// TIA Portal V17 program export: 1 tag tables, 17 data types, 25 data blocks, 3 code blocks (in call order from the OBs), 2 instance data blocks

VAR_GLOBAL   // PLC tag table "Default tag table"
   System_Byte AT %MB1000 : Byte;
   FirstScan AT %M1000.0 : Bool;
   DiagStatusUpdate AT %M1000.1 : Bool;
   AlwaysTRUE AT %M1000.2 : Bool;
   AlwaysFALSE AT %M1000.3 : Bool;
   Clock_Byte AT %MB1001 : Byte;
   Clock_10Hz AT %M1001.0 : Bool;
   Clock_5Hz AT %M1001.1 : Bool;
   "Clock_2.5Hz" AT %M1001.2 : Bool;
   Clock_2Hz AT %M1001.3 : Bool;
   "Clock_1.25Hz" AT %M1001.4 : Bool;
   Clock_1Hz AT %M1001.5 : Bool;
   "Clock_0.625Hz" AT %M1001.6 : Bool;
   "Clock_0.5Hz" AT %M1001.7 : Bool;
   TestReceive AT %M0.0 : Bool;
   ProductIn_Mem AT %M2.0 : LInt;
   GitTest AT %M0.1 : Bool;
END_VAR

TYPE "Speed_Change_Parameters"
// stored: IsFailsafeCompliant false
   STRUCT
      LabelSpeed : Int;   // Etikett hastighet
      IndexWheelVelocity : LReal;   // Indexhjul Hastighet
      IndexWheelAcceleration : LReal;   // Indexhjul Acceleration
      IndexWheelDeceleration : LReal;   // Indexhjul Decceration
      IndexWheelJerk : LReal;   // Indexhjul Jerk
   END_STRUCT;
END_TYPE

TYPE "UDT_Subsystem_Utility"
// stored: IsFailsafeCompliant false
   STRUCT
      Lifebit : Bool;   // Lifebit 1Hz, Check data exchange
      Fault : Bool;   // General Fault
      active : Bool;   // Machine is running or ready
      in_progress : Bool;   // Operation in is progress, motors are running
      EStop : Bool;   // Emergency stop active (1=good)
      General05 : Bool;   // General Signal, Operation mode 05
      General06 : Bool;   // General Signal, Operation mode 06
      General07 : Bool;   // General Signal, Operation mode 07
      General08 : Bool;   // General Signal, Operation mode 08
      General09 : Bool;   // General Signal, Operation mode 09
      General10 : Bool;   // General Signal, Operation mode 10
      General11 : Bool;   // General Signal, Operation mode 11
      General12 : Bool;   // General Signal, Operation mode 12
      General13 : Bool;   // General Signal, Operation mode 13
      General14 : Bool;   // General Signal, Operation mode 14
      General15 : Bool;   // General Signal, Operation mode 15
      Status00 : Bool;   // Motor running, status 00
      Status01 : Bool;   // Motor running, status 01
      Status02 : Bool;   // Motor running, status 02
      Status03 : Bool;   // Motor running, status 03
      Status04 : Bool;   // Motor running, status 04
      Status05 : Bool;   // Motor running, status 05
      Status06 : Bool;   // Motor running, status 06
      Status07 : Bool;   // Motor running, status 07
      Status08 : Bool;   // Motor running, status 08
      Status09 : Bool;   // Motor running, status 09
      Status10 : Bool;   // Motor running, status 10
      Status11 : Bool;   // Motor running, status 11
      Status12 : Bool;   // Motor running, status 12
      Status13 : Bool;   // Motor running, status 13
      Status14 : Bool;   // Motor running, status 14
      Status15 : Bool;   // Motor running, status 15
      Status16 : Bool;   // Motor running, status 16
      Status17 : Bool;   // Motor running, status 17
      Status18 : Bool;   // Motor running, status 18
      Status19 : Bool;   // Motor running, status 19
      Status20 : Bool;   // Motor running, status 20
      Status21 : Bool;   // Motor running, status 21
      Status22 : Bool;   // Motor running, status 22
      Status23 : Bool;   // Motor running, status 23
      Status24 : Bool;   // Motor running, status 24
      Status25 : Bool;   // Motor running, status 25
      Status26 : Bool;   // Motor running, status 26
      Status27 : Bool;   // Motor running, status 27
      Status28 : Bool;   // Motor running, status 28
      Status29 : Bool;   // Motor running, status 29
      Status30 : Bool;   // Motor running, status 30
      Status31 : Bool;   // Motor running, status 31
      Alarm000 : Bool;   // Alarm 0 active
      Alarm001 : Bool;   // Alarm 1 active
      Alarm002 : Bool;   // Alarm 2 active
      Alarm003 : Bool;   // Alarm 3 active
      Alarm004 : Bool;   // Alarm 4 active
      Alarm005 : Bool;   // Alarm 5 active
      Alarm006 : Bool;   // Alarm 6 active
      Alarm007 : Bool;   // Alarm 7 active
      Alarm008 : Bool;   // Alarm 8 active
      Alarm009 : Bool;   // Alarm 9 active
      Alarm010 : Bool;   // Alarm 10 active
      Alarm011 : Bool;   // Alarm 11 active
      Alarm012 : Bool;   // Alarm 12 active
      Alarm013 : Bool;   // Alarm 13 active
      Alarm014 : Bool;   // Alarm 14 active
      Alarm015 : Bool;   // Alarm 15 active
      Alarm016 : Bool;   // Alarm 16 active
      Alarm017 : Bool;   // Alarm 17 active
      Alarm018 : Bool;   // Alarm 18 active
      Alarm019 : Bool;   // Alarm 19 active
      Alarm020 : Bool;   // Alarm 20 active
      Alarm021 : Bool;   // Alarm 21 active
      Alarm022 : Bool;   // Alarm 22 active
      Alarm023 : Bool;   // Alarm 23 active
      Alarm024 : Bool;   // Alarm 24 active
      Alarm025 : Bool;   // Alarm 25 active
      Alarm026 : Bool;   // Alarm 26 active
      Alarm027 : Bool;   // Alarm 27 active
      Alarm028 : Bool;   // Alarm 28 active
      Alarm029 : Bool;   // Alarm 29 active
      Alarm030 : Bool;   // Alarm 30 active
      Alarm031 : Bool;   // Alarm 31 active
      Alarm032 : Bool;   // Alarm 32 active
      Alarm033 : Bool;   // Alarm 33 active
      Alarm034 : Bool;   // Alarm 34 active
      Alarm035 : Bool;   // Alarm 35 active
      Alarm036 : Bool;   // Alarm 36 active
      Alarm037 : Bool;   // Alarm 37 active
      Alarm038 : Bool;   // Alarm 38 active
      Alarm039 : Bool;   // Alarm 39 active
      Alarm040 : Bool;   // Alarm 40 active
      Alarm041 : Bool;   // Alarm 41 active
      Alarm042 : Bool;   // Alarm 42 active
      Alarm043 : Bool;   // Alarm 43 active
      Alarm044 : Bool;   // Alarm 44 active
      Alarm045 : Bool;   // Alarm 45 active
      Alarm046 : Bool;   // Alarm 46 active
      Alarm047 : Bool;   // Alarm 47 active
      Alarm048 : Bool;   // Alarm 48 active
      Alarm049 : Bool;   // Alarm 49 active
      Alarm050 : Bool;   // Alarm 50 active
      Alarm051 : Bool;   // Alarm 51 active
      Alarm052 : Bool;   // Alarm 52 active
      Alarm053 : Bool;   // Alarm 53 active
      Alarm054 : Bool;   // Alarm 54 active
      Alarm055 : Bool;   // Alarm 55 active
      Alarm056 : Bool;   // Alarm 56 active
      Alarm057 : Bool;   // Alarm 57 active
      Alarm058 : Bool;   // Alarm 58 active
      Alarm059 : Bool;   // Alarm 59 active
      Alarm060 : Bool;   // Alarm 60 active
      Alarm061 : Bool;   // Alarm 61 active
      Alarm062 : Bool;   // Alarm 62 active
      Alarm063 : Bool;   // Alarm 63 active
      Alarm064 : Bool;   // Alarm 64 active
      Alarm065 : Bool;   // Alarm 65 active
      Alarm066 : Bool;   // Alarm 66 active
      Alarm067 : Bool;   // Alarm 67 active
      Alarm068 : Bool;   // Alarm 68 active
      Alarm069 : Bool;   // Alarm 69 active
      Alarm070 : Bool;   // Alarm 70 active
      Alarm071 : Bool;   // Alarm 71 active
      Alarm072 : Bool;   // Alarm 72 active
      Alarm073 : Bool;   // Alarm 73 active
      Alarm074 : Bool;   // Alarm 74 active
      Alarm075 : Bool;   // Alarm 75 active
      Alarm076 : Bool;   // Alarm 76 active
      Alarm077 : Bool;   // Alarm 77 active
      Alarm078 : Bool;   // Alarm 78 active
      Alarm079 : Bool;   // Alarm 79 active
      Alarm080 : Bool;   // Alarm 80 active
      Alarm081 : Bool;   // Alarm 81 active
      Alarm082 : Bool;   // Alarm 82 active
      Alarm083 : Bool;   // Alarm 83 active
      Alarm084 : Bool;   // Alarm 84 active
      Alarm085 : Bool;   // Alarm 85 active
      Alarm086 : Bool;   // Alarm 86 active
      Alarm087 : Bool;   // Alarm 87 active
      Alarm088 : Bool;   // Alarm 88 active
      Alarm089 : Bool;   // Alarm 89 active
      Alarm090 : Bool;   // Alarm 90 active
      Alarm091 : Bool;   // Alarm 91 active
      Alarm092 : Bool;   // Alarm 92 active
      Alarm093 : Bool;   // Alarm 93 active
      Alarm094 : Bool;   // Alarm 94 active
      Alarm095 : Bool;   // Alarm 95 active
      Alarm096 : Bool;   // Alarm 96 active
      Alarm097 : Bool;   // Alarm 97 active
      Alarm098 : Bool;   // Alarm 98 active
      Alarm099 : Bool;   // Alarm 99 active
      Alarm100 : Bool;   // Alarm 100 active
      Alarm101 : Bool;   // Alarm 101 active
      Alarm102 : Bool;   // Alarm 102 active
      Alarm103 : Bool;   // Alarm 103 active
      Alarm104 : Bool;   // Alarm 104 active
      Alarm105 : Bool;   // Alarm 105 active
      Alarm106 : Bool;   // Alarm 106 active
      Alarm107 : Bool;   // Alarm 107 active
      Alarm108 : Bool;   // Alarm 108 active
      Alarm109 : Bool;   // Alarm 109 active
      Alarm110 : Bool;   // Alarm 110 active
      Alarm111 : Bool;   // Alarm 111 active
      Alarm112 : Bool;   // Alarm 112 active
      Alarm113 : Bool;   // Alarm 113 active
      Alarm114 : Bool;   // Alarm 114 active
      Alarm115 : Bool;   // Alarm 115 active
      Alarm116 : Bool;   // Alarm 116 active
      Alarm117 : Bool;   // Alarm 117 active
      Alarm118 : Bool;   // Alarm 118 active
      Alarm119 : Bool;   // Alarm 119 active
      Alarm120 : Bool;   // Alarm 120 active
      Alarm121 : Bool;   // Alarm 121 active
      Alarm122 : Bool;   // Alarm 122 active
      Alarm123 : Bool;   // Alarm 123 active
      Alarm124 : Bool;   // Alarm 124 active
      Alarm125 : Bool;   // Alarm 125 active
      Alarm126 : Bool;   // Alarm 126 active
      Alarm127 : Bool;   // Alarm 127 active
      OperatingHours : DWord;   // Operating hours of machine
      DownTimeHours : DWord;   // Downtime hours of machine
      Speed : Word;   // Production speed
      Container_total : DWord;   // Container counter of the actual batch.
      Container_good : DWord;   // Good container counter
      Container_reject : DWord;   // rejected container counter
      Counter_06 : DWord;   // Counter 06
      Counter_07 : DWord;   // Counter 07
      Counter_08 : DWord;   // Counter 08
      Counter_09 : DWord;   // Counter 09
      Counter_10 : DWord;   // Counter 10
      Counter_11 : DWord;   // Counter 11
      Total_Amount : Real;   // Total filling amount of the actual batch. [kg]
      Amount_01 : Real;   // Amount 01
      Amount_02 : Real;   // Amount 02
      Amount_03 : Real;   // Amount 03
      FormatName : String[20];
   END_STRUCT;
END_TYPE

TYPE "DataFromHSM"
// stored: IsFailsafeCompliant false
   STRUCT
      Sts : Struct
         xStop : Bool;   // Setzt den Spender in Stopp
         xRun : Bool;   // Setzt den Spender in Run
         xService : Bool;
         xTeach : Bool;
         xFeed : Bool;
         xConfigurationSave : Bool;
         xConfigurationLoad : Bool;
         xReceiveConfiguration : Bool;
         xCParameterSend : Bool;   // Schreibt alle über Kparam Maske ausgewählten Kparameter auf die ACP
         xCParameterReceive : Bool;   // Schreibt alle über Kparam Maske ausgewählten Kparameter in den DB
         xMparameterSend : Bool;   // Schreibt alle über Mparam Maske ausgewählten Mparameter auf die ACP
         xMparameterReceive : Bool;   // Schreibt alle über Mparam Maske ausgewählten parameter auf die DB
         xReserved : Bool;
         xGetTime : Bool;
         xGet_MAC_FW_version : Bool;
         xStatusContinuouslyTransmitted : Bool;   // 1: Aktiviert die kontinuierliche übertragung des Control Registers
         xCommunicationMonitoring : Bool;
         "x AcknowledgeFaultFromExternal" : Bool;
         xBlockProductSensor : Bool;   // 1: Produktsensor ist nicht aktiv, d.h. es wird kein Etikettierimpuls ausgelöst
         xSplice_Start : Bool;
         xReserved_25 : Bool;
         xReserved_24 : Bool;
         xReserved_23 : Bool;
         xReserved_22 : Bool;
         xReserved_21 : Bool;
         xReserved_20 : Bool;
         xReserved_19 : Bool;
         xReserved_18 : Bool;
         xReserved_17 : Bool;
         xReserved_16 : Bool;
         xReserved_15 : Bool;
         xReserved_14 : Bool;
         xDeviceStatusOK : Bool;
         xDeviceStatusWarning : Bool;
         xDeviceStatusAlarm : Bool;
         xPauseRun : Bool;
         xPauseStandby : Bool;
         xPauseService : Bool;
         xLampAlarm : Bool;
         xLampOK : Bool;
         xLampWarning : Bool;
         "xIO-Warning" : Bool;
         "xIO-Ready" : Bool;
         "xIO-Sync" : Bool;
         xSync2 : Bool;
         xSync3 : Bool;
         xLabelSensor : Bool;
         xProductSensorPolarity : Bool;
         xLowLabelSensor : Bool;
         xWebBreakSensor : Bool;
         xExternalStart : Bool;
         xSpliceActive : Bool;
         xReserved_12 : Bool;
         xReserved_11 : Bool;
         xReserved_10 : Bool;
         xReserved_09 : Bool;
         xReserved_08 : Bool;
         xReserved_07 : Bool;
         xReserved_06 : Bool;
         xReserved_05 : Bool;
         xReserved_04 : Bool;
         xReserved_03 : Bool;
         xReserved_02 : Bool;
         xReserved_01 : Bool;
         iLabelCounter : Int;
         iCounterRemaining : Int;
         iMcurr : Int;   // Status- Mittlerer Motorstrom in %
         wExtEncoder : Word;   // Status- Zählerwert des Ext. Encoders
         wErrorCode : Word;   // Fehlerwert
         wWarnNr : Word;   // Warnungscodes
         iReserved_W1 : Int;
         iReserved_W2 : Int;
         iReserved_W3 : Int;
         iReserved_W4 : Int;
         iReserved_W5 : Int;
         iReserved_W6 : Int;
      END_STRUCT;
      Cfg : Struct
         iLabellingSpeed : Int;   // in 1/10 m/min
         iTriggerDelay : Int;   // in 1/10 mm
         iLabelPosition : Int;   // in 1/10 mm
         iLabelLenght : Int;   // in mm
         iLabelGap : Int;   // in 1/10 mm
         iLabelsBurst : Int;   // 1=Aus, 2=zweimal … (mehrere Etiketten mit einem Triggerimpuls)
         iDistanceBetweenLabels : Int;   // in 1/10 mm (Abstand zwischen den Etiketten wenn mehrere pro Trigger)
         iMaxNumberOfLabelsToSkip : Int;   // 0 - n
         iTriggerBlank : Int;   // in mm
         iAccelerationRamp : Int;   // in 1/10 mm
         iSpeedInternalEncoder : Int;   // 0 = Intern, 1 = Drehgeber
         iStopRamp : Int;   // in % (Verhältnis zur Startrampe)
         iSyncOutputDelay : Int;   // in 1/10 mm
         iSyncOutputLength : Int;   // in 1/10 mm
         iSyncOutputDelay2 : Int;   // in 1/10 mm
         iSyncOutputLenght_2 : Int;   // in 1/10 mm
         iSyncOutputDelay_3 : Int;   // in 1/10 mm
         iSyncOutputLenght_3 : Int;   // in 1/10 mm
         iPreFeed : Int;   // in 1/10 mm
         iConveyorSpeed_1 : Int;
         iConveyorSpeed_2 : Int;
         iReserved_11 : Int;
         iReserved_10 : Int;
         iReserved_09 : Int;
         iReserved_08 : Int;
         iReserved_07 : Int;
         iReserved_06 : Int;
         iReserved_05 : Int;
         iReserved_04 : Int;
         iReserved_03 : Int;
         iReserved_02 : Int;
         iReserved_01 : Int;
      END_STRUCT;
      M_Par : Struct
         iSpeedInternalEncoder : Int;   // 0 = Fixed internally, 1 = Encoder fixed, 2 = Value from configuration
         iEncoderMMPerRevolution : Int;   // in 1/10 mm
         iEncoderPulsesPerRevolution : Int;   // in Pulse
         iMaximumSpeed : Int;   // in 1/10 m/min
         iInstallationMode : Int;   // 0 = normal, 1 = feed also via start button, 2 = feed with fixed length via start button, 3 = feed always with fixed length
         iLabelLengthInMMPerMotorRevolution : Int;   // in 1/100 mm
         iDistanceGapSensorToDispensingEdge : Int;   // in 1/10 mm
         iProductSensorPolarity : Int;   // 0 = NPN, 1 = NPN inverted, 2 = PNP inverted, 3 = PNP
         iSkipMode_1 : Int;   // 0 = value from configuration, 1 = value from machine parameters, 2 = end detect
         iMaxLabelSkip : Int;   // 0 - n
         iAccelerationMode : Int;   // 0 = value from configuration, 1 = value from machine parameters
         iAcceleration : Int;   // in 1/10 mm
         iGapSensor : Int;   // 0 = leading edge, 1 = trailing edge label
         iMaxCalibrationLength : Int;   // in 1/10mm
         iDecelarationMode : Int;   // 0 = value from configuration, 1 = value from machine parameters
         iDecelaration : Int;   // in % (of acceleration distance)
         iExernalStart : Int;   // 0 = off 1 = edge controlled 2 = pulse controlled
         iLowLabelInput : Int;   // 0= Off 1=On
         iBeltInput_1 : Int;   // 0= Off 1=On
         iSyncParameter_1 : Int;   // 0 = value from configuration, 1 = value from machine parameters
         iSyncOutputDelay : Int;   // in 1/10mm
         iSyncOutputLength : Int;   // in 1/10mm
         iZeroDownTimeMode_1 : Int;   // 0 = off 1 = master 2 = slave
         iZeroDownTimeSensorDistance : Int;   // in mm
         iLabelLengthInCaseOfErrorOnLowLabelSensor : Int;   // in m
         iLowLabelSensorPolarity : Int;   // 2 = PNP inverted 3 = PNP
         iWebBreakSensorPolarity : Int;   // 2 = PNP inverted 3 = PNP
         iWarningOutputPolarity_1 : Int;   // 2 = PNP inverted 3 = PNP
         iSync2Parameter_1 : Int;   // 0 = value from configuration, 1 = value from machine parameters
         iSync2OutputDelay_1 : Int;   // in 1/10mm
         iSync2OutputPulseLength_1 : Int;   // in 1/10mm
         iSync3Parameter_1 : Int;   // 0 = value from configuration, 1 = value from machine parameters
         iSync3OutputDelay_1 : Int;   // in 1/10mm
         iSync3OutputPulseLength_1 : Int;   // in 1/10mm
         iTeachTolerance : Int;   // in 1/100mm
         iSynch1Mode_1 : Int;   // 0 = production sensor 1 = trigger sensor 2 = reserve 3 = end of dispensing
         iSynch2Mode_1 : Int;   // 0 = production sensor 1 = trigger sensor 2 = reserve 3 = end of dispensing
         iSynch3Mode_1 : Int;   // 0 = production sensor 1 = trigger sensor 2 = reserve 3 = end of dispensing
         iOvercurrentCorrection : Int;   // in %
         iServiceFeedSpeed : Int;   // in 1/10 m/min
         iPreDispensingMode : Int;   // 0 = value from configuration, 1 = value from machine parameters
         iPreDispensingLength : Int;   // in 1/10 mm
         iLabelSensorWindowPreDispensingPath : Int;   // in 1/10 mm
         iLabelSensorCount : Int;
         "iSPS-Mode_1" : Int;   // 0 = Off 1 = S7 communication / 0= Off 1= S7-communication, 2 = S7-communication double size
         iZdtWin_1 : Int;   // Zero down time window mm / Zero Down Time Window mm
         iDistRes_1 : Int;   // Resolution label spacing
         "iSPS-DB-NoCtrl_1" : Int;   // SPS-DB-Nr Control (SPS->ACP) / Data block for PLC communication
         "iSPS-DB-NoStat_1" : Int;   // SPS-DB-Nr Status (ACP->SPS) / Data block for PLC communication
         iSignalFormat_1 : Int;   // Status-Server: Signalform / Is relevant for the WEBER-TOOL
         iLowLabDiam_1 : Int;   // Roll diameter for LowLabel in 1/10 mm / Roll diameter for LowLab in 1/10 mm
         iCoreDiameter_1 : Int;   // Core diameter in 1/10 mm
         iWebBreakRest_1 : Int;   // Rest after WebBreak in mm
         iLeverSetup_1 : Int;   // Do not use here / To the TEACH of the dancer position
         iLeverMinPos_1 : Int;   // Analog value angle sensor unwinder dancer Min.Pos.
         iLeverMaxPos_1 : Int;   // Analog value angle sensor unwinder dancer Max.Pos.
         "iUW-BufLength_1" : Int;   // Label path in mm between dancers min / max
         iTwinLabelMd_1 : Int;   // Double Label Mode / Double Label mode
         iLabelQueTolerans : Int;   // Setting the tolerance "Number of labels between peel bar and label sensor".
         iResetEvents : Int;   // Reset the operating data EV#007 „Number of all spent labels“ or EV#008 „Display of label roll dispensed“. 0 = off, 1 = reset EV#007 Label feeds, 2 = reset EV#008 Label meters.
         iMaintenanceDistanceKm : Int;   // Setting the maintenance interval depending on the the label roll length. [km]
         iMaintenanceDays : Int;   // Setting the maintenance interval depending on the operation time. [days]
         iProductSensorMode : Int;   // Defines the linkage of the product sensors 1 and 2 with respect to the trigger signal. 0 = Off, 1 = AND Operation (both sensors must recieve a signal), 2 = OR operation (only one sensor have to recieve a signal)
         iRewinderDiameterWarning : Int;   // Defines the diameter of the carrier web, after which a pre-warning for the rewinder is avti-vated. The following message appears "Rewinder almost full".
         arrayFirmwareVersion_1 : Array[0..19] of Char;   // Defines the diameter of the carrier web, after which the labeler stops. The following mes-sage appears "Rewinder full".
         "arrayCfg_MAC-Adress_1" : Array[0..19] of Char;   // Defines the value for the motor current, after which the following message appears "Load approaching the upper limit".
         iRewinderDiameterFull : Int;   // Parameter for activating contour mode. When the parameter is activated, the two parameters "Start contour" and "Stop contour" are displayed in the configuration menu. At the same time, the "Ramp" parameter is ignored.
         iMotorLoadLimit : Int;   // Determines the number of encoder pulses per millimeter of label path and synchronizes an optional printer at the AUX socket.
         iCountorRamp : Int;   // This Parameter is used to set the communication with different PLC versions.
         iEncoderOutPulsMM : Int;   // This parameter is used to set the distance (duration) in splice mode. The label web is ad-vanced with the reduced speed specified in parameter 071. 0 - 9999. Adjusting the value in [mm]
         iSPS_RackAndSlot : Int;   // This parameter is only used if parameter 070 is active. It is used to reduce reduce the speed in the slice mode and is calculated on the basis of the current speed. 10 - 100. Adjusting the value in [%]
         iSpliceDistance : Int;   // This parameter is only used for alternating operation and defines the transfer reserve that is still to be dispensed in alternating operation. Must be less than or equal to Par.25 RestLowLabel. 0.0 – 90.0. Adjusting the value in [m]
         iSpliceSpeedReduction : Int;   // Offset setting for operation with rotary encoder. The feed rate of the dispenser is factor Par.73 x encoder speed. 20.0 - 500.0. Adjusting the value in [%].
         iDownstream : Int := 20;   // Setting of the start ramp setting in m/s2. If the value is 0, the ramp length is used to calcu-late the acceleration. The stop ramp is set exactly as before via the ratio to the start ramp. 0.0 - 90.0. In [m/s2]
         iSpeedFactor : Int := 1000;   // Setting of a speed offset in 1/10 m/min. Only applies to the internal speed. Parameter 073 can be used in encoder mode. -20.0 - 20.0. in [%]
         iAcceleration_1 : Int := 0;   // Determines whether the material transport error "Materialtransportoffen" is to be output. The signal for the error must be applied to X22.4. 0 = Off. 1 = Error at 24V. 2 = Error at 0V.
         iSpeedOffset : Int := 0;   // Offset setting of the encoder speed for the internal calculation of Alpha HSM, e.g. for win-ding tape operation and ZDT application. Alpha HSM must calculate with baseband speed for the function of the ZDT, but dispenses with encoder speed from the winding belt. 20.0 - 500.0. In [%]
         iMaterialTransportErrorMode : Int := 0;   // Determines whether the material transport error "Materialtransportoffen" is to be output. The signal for the error must be applied to X22.4. 0 = Off. 1 = Error at 24V. 2 = Error at 0V.
         iEncoderFactor : Int := 1000;   // Offset setting of the encoder speed for the internal calculation of Alpha HSM, e.g. for win-ding tape operation and ZDT application. Alpha HSM must calculate with baseband speed for the function of the ZDT, but dispenses with encoder speed from the winding belt. 20.0 - 500.0. In [%]
         iReserve_1 : Int;
         iReserve_2 : Int;
         iReserve_3 : Int;
         iReserve_4 : Int;
         iReserve_5 : Int;
         iReserve_6 : Int;
         iReserve_7 : Int;
         iReserve_8 : Int;
         iReserve_9 : Int;
         iReserve_10 : Int;
         iReserve_11 : Int;
         iReserve_12 : Int;
         iReserve_13 : Int;
         iReserve_14 : Int;
         iReserve_15 : Int;
         iReserve_16 : Int;
         iReserve_17 : Int;
         iReserve_18 : Int;
         iReserve_19 : Int;
         iReserve_20 : Int;
         iReserve_21 : Int;
         iReserve_22 : Int;
         iReserve_23 : Int;
         iReserve_24 : Int;
         iReserve_25 : Int;
         iReserve_26 : Int;
         iReserve_27 : Int;
         iReserve_28 : Int;
         iReserve_29 : Int;
         iReserve_30 : Int;
         iReserve_31 : Int;
         iReserve_32 : Int;
         iReserve_33 : Int;
         iReserve_34 : Int;
         iReserve_35 : Int;
         iReserve_36 : Int;
         iReserve_37 : Int;
         iReserve_38 : Int;
         iReserve_39 : Int;
         iReserve_40 : Int;
         iReserve_41 : Int;
         iReserve_42 : Int;
         iReserve_43 : Int;
         iReserve_44 : Int;
         iReserve_45 : Int;
         iReserve_46 : Int;
         iReserve_47 : Int;
         iReserve_48 : Int;
         iReserve_49 : Int;
         iReserve_50 : Int;
         iReserve_51 : Int;
      END_STRUCT;
   END_STRUCT;
END_TYPE

TYPE "DataToHSM"
// stored: IsFailsafeCompliant false
   STRUCT
      Cmd : Struct   // Command Send
         xStop : Bool;   // Offline
         xRun : Bool;   // Online
         xService : Bool;
         xTeach : Bool;
         xFeed : Bool;
         xSaveConfiguration : Bool;   // Reserved but not used for the time being
         xLoadConfiguration : Bool;   // Reserved but not used for the time being
         xRecieveContent : Bool;   // Reserved but not used for the time being
         xCparameterSend : Bool;   // Starts sending all K parameters selected via Kparameter mask to the labeling system / Starts sending all C parameters selected via C parameter mask to the labeling system
         xCparameterReceive : Bool;   // Requests the labeling system to send all parameters
         xMparameterSend : Bool;   // Starts sending all the M parameters selected via the Mparameter mask to the labeling system
         xMparameterReceive : Bool;   // Requests all labeling parameters to be sent from the labeling system
         xReserve : Bool;
         xReceiveTime : Bool;
         xGetMACandFWversion : Bool;
         xActivateContinuousStatus : Bool;   // 1: Activates the continuous transfer of the control register (initially not used)
         xWatchDog : Bool;   // Sign of Life Bit
         xAcknowledgeFaultFromExternal : Bool;   // PLC can directly acknowledge a malfunction of the labeling system
         xBlockProductPhotocell : Bool;   // 1: Product sensor is not active, i.e. no labeling pulse is triggered
         "xSplice-Start" : Bool;
         xReserved_19 : Bool;
         xReserved_18 : Bool;
         xReserved_17 : Bool;
         xReserved_16 : Bool;
         xReserved_15 : Bool;
         xReserved_14 : Bool;
         xReserved_13 : Bool;
         xReserved_12 : Bool;
         xReserved_11 : Bool;
         xReserved_10 : Bool;
         xReserved_09 : Bool;
         xReserved_08 : Bool;
         ParaMask : "HSMConfigAndMachineParameterMask";
         iUpdateRate : Int;   // Rate in ms at which the control register is updated
         iReserved_03 : Int;
         iReserved_02 : Int;
         iReserved_01 : Int;
      END_STRUCT;
      Cfg : Struct   // Configuration Parameters Send
         iDesiredInternalSpeed : Int;   // in 1/10 m / min (desired speed value)
         iDispenseDelay : Int;   // in 1/10 mm
         iLabelPosition : Int;   // in 1/10 mm
         iLabelLength : Int;   // in mm
         iLabelGap : Int;   // in 1/10 mm
         iLabelBurst : Int;   // 1 = off, 2 = twice ... (several labels with one trigger pulse)
         iLabelDistance : Int;   // in 1/10 mm (distance between the labels if several per trigger)
         iMaxNumberOfLabelSkips : Int;   // 0 - n
         iTriggerBlanking : Int;   // in mm
         iAccelerationRamp : Int;   // in 1/10 mm
         iSpeedInternalOrEncoder : Int;   // 0 = internal, 1 = encoder
         iStopRamp : Int;   // in% (ratio to acceleration ramp)
         iSyncOutputDelay : Int;   // in 1/10 mm
         iSyncOutputLenght : Int;   // in 1/10 mm
         iSyncOutput2Delay : Int;   // in 1/10 mm
         iSyncOutput2Lenght : Int;   // in 1/10 mm
         iSyncOutput3Delay : Int;   // in 1/10 mm
         iSyncOutput3Lenght : Int;   // in 1/10 mm
         iPreFeedLenght : Int;   // in 1/10 mm
         iConveyorSpeed_1 : Int;
         iConveyorSpeed_2 : Int;
         iReserved_11 : Int;
         iReserved_10 : Int;
         iReserved_09 : Int;
         iReserved_08 : Int;
         iReserved_07 : Int;
         iReserved_06 : Int;
         iReserved_05 : Int;
         iReserved_04 : Int;
         iReserved_03 : Int;
         iReserved_02 : Int;
         iReserved_01 : Int;
      END_STRUCT;
      MPar : Struct   // Machine Parameters Send
         iSpeedInternalOrEncoder : Int;   // 0 = Fixed internally, 1 = Encoder fixed, 2 = Value from configuration
         iDistancePerEncoderRevolution : Int;   // in 1/10 mm
         iPulsesPerEncoderRevolution : Int;   // in Pulse
         iMaxSpeed : Int;   // in 1/10 m/min
         iInstallationsMode : Int;   // 0 = normal, 1 = feed also via start button, 2 = feed with fixed length via start button, 3 = feed always with fixed length
         iBackingPaperLengthPerMotorRevolution : Int;   // in 1/100 mm
         iDistanceToDispensingEdgeToGapSensor : Int;   // in 1/10 mm (required for changeable dispense tongues and changed depending on the product)
         iProductsensorPolarity : Int;   // 0 = NPN, 1 = NPN inverted, 2 = PNP inverted, 3 = PNP
         iSkipMode : Int;   // 0 = value from configuration, 1 = value from machine parameters, 2 = end detect
         iMaxNumberOfLabelSkips : Int;   // 0 - n
         iAccelerationRampMode : Int;   // 0 = value from configuration, 1 = value from machine parameters
         iAccelerationRamp : Int;   // in 1/10 mm
         iGapSensor : Int;   // 0 = leading edge, 1 = trailing edge label
         iMaxCalibrationDistance : Int;   // in 1/10mm
         iDecelerationRampMode : Int;   // 0 = value from configuration, 1 = value from machine parameters
         iDecelerationRamp : Int;   // in% (ratio to acceleration ramp)
         iExternalStart : Int;   // 0 = off 1 = edge controlled 2 = pulse controlled
         iLowLabelInput : Int;   // 0 = off 1 = on
         iRibbonInput : Int;   // 0 = off 1 = on
         iSyncParameter : Int;   // 0 = value from configuration, 1 = value from machine parameters
         iSyncOutputDelay : Int;   // in 1/10mm
         iSyncOutputLenght : Int;   // in 1/10mm
         iZeroDownTimeMode : Int;   // 0 = Off 1 = Master 2 = Slave
         iZeroDownTimeSensorDistance : Int;   // in mm
         iRestLenghtOnLowLabel : Int;   // in m
         iLowLabelSensorPolarity : Int;   // 2 = PNP inverted 3 = PNP
         iWebBreakSensorPolarity : Int;   // 2 = PNP inverted 3 = PNP
         iWarningOutputPolarity : Int;   // 2 = PNP inverted 3 = PNP
         iSync2Parameter : Int;   // 0 = value from configuration, 1 = value from machine parameters
         iSync2OutputDelay : Int;   // in 1/10mm
         iSync2OutputLenght : Int;   // in 1/10mm
         iSync3Parameter : Int;   // 0 = value from configuration, 1 = value from machine parameters
         iSync3OutputDelay : Int;   // in 1/10mm
         iSync3OutputLenght : Int;   // in 1/10mm
         iTeachTolerance : Int;   // in 1/100mm
         iSynch1Mode : Int;   // 0 = production sensor 1 = trigger sensor 2 = reserve 3 = end of dispense
         iSynch2Mode : Int;   // 0 = production sensor 1 = trigger sensor 2 = reserve 3 = end of dispense
         iSynch3Mode : Int;   // 0 = production sensor 1 = trigger sensor 2 = reserve 3 = end of dispense
         iOverCurrentCorrection : Int;   // in %
         iServiceFeedRate : Int := 10;   // in 1/10 m/min
         iPreFeedMode : Int;   // 0 = value from configuration, 1 = value from machine parameters
         iPreFeed : Int;   // in 1/10 mm
         iLabelSensorWindowPreFeedLenght : Int;   // in 1/10 mm
         iLabelSensorCount : Int;
         "iSPS-Mode" : Int;   // 0= Off 1= S7-Kommunikation / 0= Off 1= S7-communication, 2 = S7-communication double size
         iZdtWin : Int;   // Zero Down Time Window mm
         iDistRes : Int;   // Resolution label spacing
         "iSPS-DB-No-Ctrl" : Int;   // Data block for PLC communication
         "iSPS-DB-No-Stat" : Int;   // Data block for PLC communication
         iSignalFormat : Int;   // Is relevant for the WEBER-TOOL
         iLowLabDiam : Int;   // Roll diameter for LowLab in 1/10 mm
         iCoreDiameter : Int;   // Core diameter in 1/10 mm
         iWebBreakRest : Int;   // Rest after WebBreak in mm
         iLeverSetup : Int;   // To the TEACH of the dancer position
         iLeverMinPos : Int;   // Analog value angle sensor unwinder dancer Min.Pos.
         iLeverMaxPos : Int;   // Analog value angle sensor unwinder dancer Max.Pos.
         "iUW-BufLength" : Int;   // Label path in mm between dancers min / max
         iTwinLabelMd : Int;   // Double Label mode
         iLabQueuwTolerance : Int := 10;   // Setting the tolerance "Number of labels between peel bar and label sensor".
         iResetEvents : Int;   // Reset the operating data EV#007 „Number of all spent labels“ or EV#008 „Display of label roll dispensed“. 0 = off, 1 = reset EV#007 Label feeds, 2 = reset EV#008 Label meters.
         iMaintananceDistancekm : Int;   // Setting the maintenance interval depending on the the label roll length. [km]
         iMaintananceDays : Int;   // Setting the maintenance interval depending on the operation time. [days]
         iProductSensorMode : Int;   // Defines the linkage of the product sensors 1 and 2 with respect to the trigger signal. 0 = Off, 1 = AND Operation (both sensors must recieve a signal), 2 = OR operation (only one sensor have to recieve a signal)
         iRewinderDiameterWarning : Int := 2600;   // Defines the diameter of the carrier web, after which a pre-warning for the rewinder is avti-vated. The following message appears "Rewinder almost full".
         iRewinderDiameterFull : Int := 2650;   // Defines the diameter of the carrier web, after which the labeler stops. The following mes-sage appears "Rewinder full".
         iMotorLoadLimit : Int := 90;   // Defines the value for the motor current, after which the following message appears "Load approaching the upper limit".
         iContourRamp : Int;   // Parameter for activating contour mode. When the parameter is activated, the two parameters "Start contour" and "Stop contour" are displayed in the configuration menu. At the same time, the "Ramp" parameter is ignored.
         iEncoderOutPulsPermm : Int;   // Determines the number of encoder pulses per millimeter of label path and synchronizes an optional printer at the AUX socket.
         iPLCRackAndSlot : Int := 10;   // This Parameter is used to set the communication with different PLC versions.
         iSliceDistance : Int := 2000;   // This parameter is used to set the distance (duration) in splice mode. The label web is ad-vanced with the reduced speed specified in parameter 071. 0 - 9999. Adjusting the value in [mm]
         iSpliceSpeedReduction : Int := 33;   // This parameter is only used if parameter 070 is active. It is used to reduce reduce the speed in the slice mode and is calculated on the basis of the current speed. 10 - 100. Adjusting the value in [%]
         iDownstream : Int := 20;   // This parameter is only used for alternating operation and defines the transfer reserve that is still to be dispensed in alternating operation. Must be less than or equal to Par.25 RestLowLabel. 0.0 – 90.0. Adjusting the value in [m]
         iSpeedFactor : Int := 1000;   // Offset setting for operation with rotary encoder. The feed rate of the dispenser is factor Par.73 x encoder speed. 20.0 - 500.0. Adjusting the value in [%].
         iAcceleration : Int;   // Setting of the start ramp setting in m/s2. If the value is 0, the ramp length is used to calcu-late the acceleration. The stop ramp is set exactly as before via the ratio to the start ramp. 0.0 - 90.0. In [m/s2]
         iSpeedOffset : Int;   // Setting of a speed offset in 1/10 m/min. Only applies to the internal speed. Parameter 073 can be used in encoder mode. -20.0 - 20.0. in [%]
         iMaterialTransportErrorMode : Int;   // Determines whether the material transport error "Materialtransportoffen" is to be output. The signal for the error must be applied to X22.4. 0 = Off. 1 = Error at 24V. 2 = Error at 0V.
         iEncoderFactor : Int := 1000;   // Offset setting of the encoder speed for the internal calculation of Alpha HSM, e.g. for win-ding tape operation and ZDT application. Alpha HSM must calculate with baseband speed for the function of the ZDT, but dispenses with encoder speed from the winding belt. 20.0 - 500.0. In [%]
         Reserve_1 : Int;
         Reserve_2 : Int;
         Reserve_3 : Int;
         Reserve_4 : Int;
         Reserve_5 : Int;
         Reserve_6 : Int;
         Reserve_7 : Int;
         Reserve_8 : Int;
         Reserve_9 : Int;
         Reserve_10 : Int;
         Reserve_11 : Int;
         Reserve_12 : Int;
         Reserve_13 : Int;
         Reserve_14 : Int;
         Reserve_15 : Int;
         Reserve_16 : Int;
         Reserve_17 : Int;
         Reserve_18 : Int;
         Reserve_19 : Int;
         Reserve_20 : Int;
         Reserve_21 : Int;
         Reserve_22 : Int;
         Reserve_23 : Int;
         Reserve_24 : Int;
         Reserve_25 : Int;
         Reserve_26 : Int;
         Reserve_27 : Int;
         Reserve_28 : Int;
         Reserve_29 : Int;
         Reserve_30 : Int;
         Reserve_31 : Int;
         Reserve_32 : Int;
         Reserve_33 : Int;
         Reserve_34 : Int;
         Reserve_35 : Int;
         Reserve_36 : Int;
         Reserve_37 : Int;
         Reserve_38 : Int;
         Reserve_39 : Int;
         Reserve_40 : Int;
         Reserve_41 : Int;
         Reserve_42 : Int;
         Reserve_43 : Int;
         Reserve_44 : Int;
         Reserve_45 : Int;
         Reserve_46 : Int;
         Reserve_47 : Int;
         Reserve_48 : Int;
         Reserve_49 : Int;
         Reserve_50 : Int;
         Reserve_51 : Int;
      END_STRUCT;
   END_STRUCT;
END_TYPE

TYPE "HSMConfigAndMachineParameterMask"
// stored: IsFailsafeCompliant false
   STRUCT
      HSMConfig_1 : "HSMConfigParaMask1";
      HSMConfig_2 : "HSMConfigParaMask2";
      HSMMachine_1 { S7_SetPoint := 'True'} : "HSMMachineParaMask1";
      HSMMachine_2 { S7_SetPoint := 'True'} : "HSMMachineParaMask2";
      HSMMachine_3 { S7_SetPoint := 'True'} : "HSMMachineParaMask3";
      HSMMachine_4 { S7_SetPoint := 'True'} : "HSMMachineParaMask4";
      HSMMachine_5 { S7_SetPoint := 'True'} : "HSMMachineParaMask5";
      HSMMachine_6 { S7_SetPoint := 'True'} : "HSMMachineParaMask6";
      HSMMachine_7 { S7_SetPoint := 'True'} : "HSMMachineParaMask7";
      HSMMachine_8 { S7_SetPoint := 'True'} : "HSMMachineParaMask8";
   END_STRUCT;
END_TYPE

TYPE "HSM_AlarmWarning"
// stored: IsFailsafeCompliant false
   STRUCT
      WWarning_08_Rewinder_Almost_Full : Bool;   // Rewinder almost full. Do a controlled stop and change otherwise machine may stop unexpected.
      WWarning_09_Roll_End_1 : Bool;
      WWarning_10_Roll_End_2 : Bool;
      WWarning_11_Roll_End_3 : Bool;
      WWarning_12 : Bool;
      WWarning_13 : Bool;
      WWarning_14 : Bool;
      WWarning_15 : Bool;
      WWarning_00 : Bool;
      WWarning_01_Find_Rotor_Position : Bool;   // Warning Rotor Position. Try restart.
      WWarning_02 : Bool;
      WWarning_03_Number_Of_Labels_Reached : Bool;   // This message indicates that the "Countdown" function has run to the end and has reached the end value "000".
      WWarning_04_Low_Label_Reached : Bool;   // This message indicates that the pre-set minimum diameter of the label roll for optional low label warning has been reached. When the residual label length (machine parameter [025] has been entered, the labeling mode is continued until this value has been reached. Thereafter, the labeler will stop and the "Web end reached” error message will be dis-played.
      WWarning_05_ZeroDownTime_Lan_Link_timeout : Bool;
      WWarning_06_ZeroDownTime_Parameter_error : Bool;
      WWarning_07 : Bool;
      AAlarm_14_Motor_Overcurrent : Bool;   // This message implies that the strain on the motor controller by the maximum current is too high. Potential causes: Too high cycle rate, paper brake to tight, material wrapped around the drive unit. Solution: Switch off the labeler, repair fault, switch on the labeler.
      AAlarm_15_Dancer_Arm_Stop_Reached : Bool;   // Unwinder dancer arm reached end position. End of label roll.
      AAlarm_16_Rewinder_Full : Bool;   // Rewinder full. Remove backing paper from rewinder and reattach to rewinder.
      AAlarm_17_Rewinder_Web_Break : Bool;   // Backing paper (web) broke or not attached to rewinder.
      AAlarm_18 : Bool;
      AAlarm_19 : Bool;
      AAlarm_20 : Bool;
      AAlarm_21 : Bool;
      AAlarm_6 : Bool;
      AAlarm_7_Motor_Start_Error : Bool;   // This message implies that the internal zero-compensation could not be performed. Switch off the labeler at the mains switch and wait until the display has gone off. Thereafter, switch the labeler back on.
      AAlarm_8_Motor_Position_Error : Bool;   // This message indicates that the servomotor cannot determine its rotor position during the initialization phase. Switch off the labeler at the mains switch and wait until the display has gone off. Thereafter, switch the labeler back on.
      AAlarm_9_Motor_Position_Control_Error : Bool;   // This message indicates that the servomotor cannot determine its prescribed position.
      AAlarm_10_Motor_Current_Target_Not_Reached : Bool;   // This message implies that the motor overload is too high, e.g. due to a short-circuit or ex-ternal interference.
      AAlarm_11_Label_Gap_Not_Found : Bool;   // This message implies that the label sensor does not detect the label stock. The existing labels between the label sensor and dispenser are dispensed completely. Thereafter, the system is switched to "Fault" (compare section above).
      AAlarm_12_Unwinder_Web_Break : Bool;   // This message means that the optional web break sensor detects that no label material is present. The currently applied label is still applied. Thereafter, the labeler interrupts the labeling cycle. Possible causes: Web break or end of web.
      AAlarm_13_Web_End : Bool;   // This message implies that the low label warning has been triggered and the pre-programmed residual label roll length (under machine parameter [025]) has lapsed. When the value for the remaining label length is set to "0" m (default value), a warning will be output but no "Error" triggered.
   END_STRUCT;
END_TYPE

TYPE "typeFromHMI"
// stored: IsFailsafeCompliant false
   STRUCT
      xBtn_Stop : Bool;   // Stop HSM
      xBtn_Run : Bool;   // Start HSM
      xBtn_Teach : Bool;   // Calibrate label process = 1
      xBtn_Feed : Bool;   // Feed label manually
      xBtn_Get_FW_MAC : Bool;   // Get firmware version and MAC address.
      xBtn_Activate_Splice : Bool;
      xSend_Para : Bool;
      rLabel_Speed : Real := 60.0;   // Label speed
      xBtn_Save_Par : Bool;   // Save parameters to HSM
      xHSM_Active : Bool := true;   // Enabled = 1, Disabled = 0
      xGet_Parameters : Bool;
      iLabels_Per_Trigger : Int := 1;
      iTrigger_Supression : Int := 0;
      iProduct_Sensor_Polarity : Int := 3;
      iDouble_Label : Int := 0;
      iSpeed_Int_Ext : Int;
      iLabel_Length : Int := 0;
      rLabel_Position : Real := 1.0;   // Calibration offset label position on peeler plate.
      rTrig_Delay : Real := 0.0;   // Delay trigger labelling when sensor trig.
      rSpeed_Offset : Real := 0.0;   // Label speed + speed offset = speed internal
      rGap_Sensor_To_Dispenser_Tongue : Real := 240.0;
      rLabel_Spacing : Real := 2.0;
      rPre_Dispensing_Lenght : Real := 0.0;
      rLabel_Gap : Real := 0.0;
      rSpeed_Offset_Percentage : Real := 0.0;
      ConfigAndMachineParaMask : "HSMConfigAndMachineParameterMask";
   END_STRUCT;
END_TYPE

TYPE "HSMConfigParaMask1"
// stored: IsFailsafeCompliant false
   STRUCT
      iDesiredInternalSpeed : Bool;
      iDispenseDelay : Bool;
      iLabelPosition : Bool;
      iLabelLength : Bool;
      iLabelGap : Bool;
      iLabelBurst : Bool;
      iLabelDistance : Bool;
      iMaxNumberOfLabelSkips : Bool;
      iTriggerBlanking : Bool;
      iAccelerationRamp : Bool;
      iSpeedInternalOrEncoder : Bool;
      iStopRamp : Bool;
      iSyncOutputDelay : Bool;
      iSyncOutputLenght : Bool;
      iSyncOutput2Delay : Bool;
      iSyncOutput2Lenght : Bool;
   END_STRUCT;
END_TYPE

TYPE "HSMConfigParaMask2"
// stored: IsFailsafeCompliant false
   STRUCT
      iSyncOutput3Delay : Bool;
      iSyncOutput3Lenght : Bool;
      iPreFeedLenght : Bool;
      iConveyorSpeed_1 : Bool;
      iConveyorSpeed_2 : Bool;
      iReserved_1 : Bool;
      iReserved_2 : Bool;
      iReserved_3 : Bool;
      iReserved_4 : Bool;
      iReserved_5 : Bool;
      iReserved_6 : Bool;
      iReserved_7 : Bool;
      iReserved_8 : Bool;
      iReserved_9 : Bool;
      iReserved_10 : Bool;
      iReserved_11 : Bool;
   END_STRUCT;
END_TYPE

TYPE "HSMMachineParaMask1"
// stored: IsFailsafeCompliant false
   STRUCT
      iSpeedInternalOrEncoder : Bool;
      iDistancePerEncoderRevolution : Bool;
      iPulsesPerEncoderRevolution : Bool;
      iMaxSpeed : Bool;
      iInstallationsMode : Bool;
      iBackingPaperLengthPerMotorRevolution : Bool;
      iDistanceToDispensingEdgeToGapSensor : Bool;
      iProductsensorPolarity : Bool;
      iSkipMode : Bool;
      iMaxNumberOfLabelSkips : Bool;
      iAccelerationRampMode : Bool;
      iAccelerationRamp : Bool;
      iGapSensor : Bool;
      iMaxCalibrationDistance : Bool;
      iDecelerationRampMode : Bool;
      iDecelerationRamp : Bool;
   END_STRUCT;
END_TYPE

TYPE "HSMMachineParaMask2"
// stored: IsFailsafeCompliant false
   STRUCT
      iExternalStart : Bool;
      iLowLabelInput : Bool;
      iRibbonInput : Bool;
      iSyncParameter : Bool;
      iSyncOutputDelay : Bool;
      iSyncOutputLenght : Bool;
      iZeroDownTimeMode : Bool;
      iZeroDownTimeSensorDistance : Bool;
      iRestLenghtOnLowLabel : Bool;
      iLowLabelSensorPolarity : Bool;
      iWebBreakSensorPolarity : Bool;
      iWarningOutputPolarity : Bool;
      iSync2Parameter : Bool;
      iSync2OutputDelay : Bool;
      iSync2OutputLenght : Bool;
      iSync3Parameter : Bool;
   END_STRUCT;
END_TYPE

TYPE "HSMMachineParaMask3"
// stored: IsFailsafeCompliant false
   STRUCT
      iSync3OutputDelay : Bool;
      iSync3OutputLenght : Bool;
      iTeachTolerance : Bool;
      iSynch1Mode : Bool;
      iSynch2Mode : Bool;
      iSynch3Mode : Bool;
      iOverCurrentCorrection : Bool;
      iServiceFeedRate : Bool;
      iPreFeedMode : Bool;
      iPreFeed : Bool;
      iLabelSensorWindowPreFeedLenght : Bool;
      iLabelSensorCount : Bool;
      "iSPS-Mode" : Bool;
      iZdtWin : Bool;
      iDistRes : Bool;
      "iSPS-DB-No-Ctrl" : Bool;
   END_STRUCT;
END_TYPE

TYPE "HSMMachineParaMask4"
// stored: IsFailsafeCompliant false
   STRUCT
      "iSPS-DB-No-Stat" : Bool;
      iSignalFormat : Bool;
      iLowLabDiam : Bool;
      iCoreDiameter : Bool;
      iWebBreakRest : Bool;
      iLeverSetup : Bool;
      iLeverMinPos : Bool;
      iLeverMaxPos : Bool;
      "iUW-BufLength" : Bool;
      iTwinLabelMd : Bool;
      iLabQueuwTolerance : Bool;
      iResetEvents : Bool;
      iMaintananceDistancekm : Bool;
      iMaintananceDays : Bool;
      iProductSensorMode : Bool;
      iRewinderDiameterWarning : Bool;
   END_STRUCT;
END_TYPE

TYPE "HSMMachineParaMask5"
// stored: IsFailsafeCompliant false
   STRUCT
      iRewinderDiameterFull : Bool;
      iMotorLoadLimit : Bool;
      iContourRamp : Bool;
      iEncoderOutPulsPermm : Bool;
      iPLCRackAndSlot : Bool;
      iSliceDistance : Bool;
      iSpliceSpeedReduction : Bool;
      iDownstream : Bool;
      iSpeedFactor : Bool;
      iAcceleration : Bool;
      iSpeedOffset : Bool;
      iMaterialTransportErrorMode : Bool;
      iEncoderFactor : Bool;
      MPARA_I_Reserve_7 : Bool;
      MPARA_I_Reserve_8 : Bool;
      MPARA_I_Reserve_9 : Bool;
   END_STRUCT;
END_TYPE

TYPE "HSMMachineParaMask6"
// stored: IsFailsafeCompliant false
   STRUCT
      MPARA_I_Reserve_10 : Bool;
      MPARA_I_Reserve_11 : Bool;
      MPARA_I_Reserve_12 : Bool;
      MPARA_I_Reserve_13 : Bool;
      MPARA_I_Reserve_14 : Bool;
      MPARA_I_Reserve_15 : Bool;
      MPARA_I_Reserve_16 : Bool;
      MPARA_I_Reserve_17 : Bool;
      MPARA_I_Reserve_18 : Bool;
      MPARA_I_Reserve_19 : Bool;
      MPARA_I_Reserve_20 : Bool;
      MPARA_I_Reserve_21 : Bool;
      MPARA_I_Reserve_22 : Bool;
      MPARA_I_Reserve_23 : Bool;
      MPARA_I_Reserve_24 : Bool;
      MPARA_I_Reserve_25 : Bool;
   END_STRUCT;
END_TYPE

TYPE "HSMMachineParaMask7"
// stored: IsFailsafeCompliant false
   STRUCT
      MPARA_I_Reserve_26 : Bool;
      MPARA_I_Reserve_27 : Bool;
      MPARA_I_Reserve_28 : Bool;
      MPARA_I_Reserve_29 : Bool;
      MPARA_I_Reserve_30 : Bool;
      MPARA_I_Reserve_31 : Bool;
      MPARA_I_Reserve_32 : Bool;
      MPARA_I_Reserve_33 : Bool;
      MPARA_I_Reserve_34 : Bool;
      MPARA_I_Reserve_35 : Bool;
      MPARA_I_Reserve_36 : Bool;
      MPARA_I_Reserve_37 : Bool;
      MPARA_I_Reserve_38 : Bool;
      MPARA_I_Reserve_39 : Bool;
      MPARA_I_Reserve_40 : Bool;
      MPARA_I_Reserve_41 : Bool;
   END_STRUCT;
END_TYPE

TYPE "HSMMachineParaMask8"
// stored: IsFailsafeCompliant false
   STRUCT
      MPARA_I_Reserve_42 : Bool;
      MPARA_I_Reserve_43 : Bool;
      MPARA_I_Reserve_44 : Bool;
      MPARA_I_Reserve_45 : Bool;
      MPARA_I_Reserve_46 : Bool;
      MPARA_I_Reserve_47 : Bool;
      MPARA_I_Reserve_48 : Bool;
      MPARA_I_Reserve_49 : Bool;
      MPARA_I_Reserve_50 : Bool;
      MPARA_I_Reserve_51 : Bool;
      MPARA_I_Reserve_52 : Bool;
      MPARA_I_Reserve_53 : Bool;
      MPARA_I_Reserve_54 : Bool;
      MPARA_I_Reserve_55 : Bool;
      MPARA_I_Reserve_56 : Bool;
      MPARA_I_Reserve_57 : Bool;
   END_STRUCT;
END_TYPE

DATA_BLOCK "DB - Btn_HSM_Side"   // DB81
{ S7_Optimized_Access := 'FALSE' }
VERSION : 0.1
// stored: AutoNumber true, DBAccessibleFromOPCUA true, DBAccessibleFromWebserver true, IsOnlyStoredInLoadMemory false, IsWriteProtectedInAS false
   VAR RETAIN
      Teach : Bool;
      Feed : Bool;
      Start : Bool;
      Activate : Bool;
   END_VAR
BEGIN
END_DATA_BLOCK

DATA_BLOCK "DB - Btn_HSM_Zon1"   // DB82
{ S7_Optimized_Access := 'FALSE' }
VERSION : 0.1
// stored: AutoNumber true, DBAccessibleFromOPCUA true, DBAccessibleFromWebserver true, IsOnlyStoredInLoadMemory false, IsWriteProtectedInAS false
   VAR RETAIN
      Teach : Bool;
      Feed : Bool;
      Start : Bool;
      Activate : Bool;
   END_VAR
BEGIN
END_DATA_BLOCK

DATA_BLOCK "DB - Btn_HSM_Zon2"   // DB83
{ S7_Optimized_Access := 'FALSE' }
VERSION : 0.1
// stored: AutoNumber true, DBAccessibleFromOPCUA true, DBAccessibleFromWebserver true, IsOnlyStoredInLoadMemory false, IsWriteProtectedInAS false
   VAR RETAIN
      Teach : Bool;
      Feed : Bool;
      Start : Bool;
      Activate : Bool;
   END_VAR
BEGIN
END_DATA_BLOCK

DATA_BLOCK "DB - Btn_Tags"   // DB60
{ S7_Optimized_Access := 'FALSE' }
VERSION : 0.1
// stored: AutoNumber true, DBAccessibleFromOPCUA true, DBAccessibleFromWebserver true, IsOnlyStoredInLoadMemory false, IsWriteProtectedInAS false
   VAR RETAIN
      Starta_Banor : Bool;   // Starta Banor
      Reject_Topp_Pulse : Bool;   // Reject Topp
      Reject_Bottom_Pulse : Bool;   // Reject Botten
      Ignore_External_Pause : Bool;   // Ignorera External Pause
      MoveRotateProductCylinder : Bool;   // Rotera Dosa Cylinder
      Index_Wheel_Brake : Bool;   // Indexhjul Broms
      StandbyOff : Bool;   // Deaktivera Standby
      JogFunctionActive : Bool;   // Aktivera Jog
      Jog : Bool;   // Kör Jog
      Speed_1 : Bool;   // Hastighet 1
      Speed_2 : Bool;   // Hastighet 2
      Speed_3 : Bool;   // Hastighet 3
      EmptyMachine : Bool;   // Töm Maskin
      Activate_Cam1 : Bool;   // Aktivera Kamera 1
      Activate_Cam2 : Bool;   // Aktivera Kamera 2
      Activate_Cam3 : Bool;   // Aktivera Kamera 3
      Activate_Cam4 : Bool;   // Aktivera Kamera 4
      Speed_4 : Bool;   // Hastighet 4
      Speed_5 : Bool;   // Hastighet 5
      Disable_LabelAdjustMent : Bool;   // Deaktivera Etikettjustering
      Activate_Printer : Bool;   // Printer
   END_VAR
BEGIN
END_DATA_BLOCK

DATA_BLOCK "DB - Counters"   // DB27
{ S7_Optimized_Access := 'FALSE' }
VERSION : 0.1
// stored: AutoNumber true, DBAccessibleFromOPCUA true, DBAccessibleFromWebserver true, IsOnlyStoredInLoadMemory false, IsWriteProtectedInAS false
   VAR RETAIN
      Product_In : Int;
      Rejected_Total : Int;
      Rejected_Side : Int;
      Rejected_Top : Int;
      Rejected_Bottom : Int;
      Product_Out : Int;
   END_VAR
BEGIN
END_DATA_BLOCK

DATA_BLOCK "DB - Events_To_PC"   // DB26
{ S7_Optimized_Access := 'FALSE' }
VERSION : 0.1
// stored: AutoNumber true, DBAccessibleFromOPCUA true, DBAccessibleFromWebserver true, IsOnlyStoredInLoadMemory false, IsWriteProtectedInAS false
   VAR
      ADoorNotClosed : Bool;   // Door to Index Wheel not Closed
      ANoLabelGapFound : Bool;   // Kontrollera etikettladdning vid etikett givare
      ARewinderTimeOut : Bool;   // Kontrollera etikettladdning vid upprullare
      WExternalPause : Bool;   // Machine paused by external machine
      ANoLabel_In_LabelQueue : Bool;   // Ingen Etikett hittad i etikettkö
      AStopInReject : Bool;   // Product stuck in side outfeed
      ACam4_Max_Rejects_Reached : Bool;   // Cam 4 max rejects reached. Check Camera HMI.
      AE_Stop_Not_Ok : Bool;   // Safety circuit not okay. Check emergency buttons and reset.
      ALabelEndOnActiveUnwinder : Bool;   // Etikett slut
      WLabelLowUnwinder1 : Bool;   // Etikett låg avrullare 1
      WLabelLowUnwinder2 : Bool;   // Etikett låg avrullare 2
      ILabelSeamedEvent : Bool;   // Label Seamed
      ACam3_Max_Rejects_Reached : Bool;   // Camera 3 max rejects reached. Check Camera HMI
      AFeed_Label_Drive_Error : Bool;   // Fel på motor till Kö
      ADispense_Label_Drive_Error : Bool;   // Fel på motor till Etikett Dispensering
      ARotate_Product_Drive_Error : Bool;   // Fault with rotate product motor.
      AIndex_Wheel_Drive_Error : Bool;   // Fault with index wheel motor.
      ARewinder_Drive_Error : Bool;   // Fel på motor till Upprullare
      AFindLabelGap_Error : Bool;   // Fel på kommunikation mellan Dispenerings drive och PLC
      AZone2_Conveyor_Error : Bool;   // Fault Zone 2 conveyor motor
      AZone2_Queue_Error : Bool;   // Fault Zone 2 queue motor.
      AZone2_Side_HSM_Move_Error : Bool;   // Fault Zone 2 Label adjust motor.
      ARotation_Error : Bool;   // Fault with product orientation motor. Either left or right.
      AZone2_Side_HSM_Error : Bool;   // Fault Zone 2 side motors labeling.
      AZone1_Conveyor_Error : Bool;   // Fault Zone 1 conveyor motor,
      AZone1_Queue_Error : Bool;   // Fault Zone 1 queue motor.
      AZone1_Side_HSM_Error : Bool;   // Fault Zone 1 side motors labeling.
      ANo_Product_In_Index_Wheel : Bool;   // No Product in Index Wheel.
      AZone1ConveyorFull : Bool;   // Zone 1 Conveyor full of products. Clear products and start machine.
      AZone2ConveyorFull : Bool;   // Zone 2 Conveyor full of products. Clear products and start machine.
      ARewinderFull : Bool;   // Upprullaren är full
      AHSMSideNotOK : Bool;   // HSM Side is not Ready.
      AHSMZon1NotOK : Bool;   // HSM Zone 1 is not Ready.
      AHSMZon2NotOK : Bool;   // HSM Zone 2 is not Ready.
      AMachineStoppedByWatchdog : Bool;   // Machine stopped by lost connection between HMI and PLC.
      IIgnoreExternalPauseActive : Bool;   // Ignore External Pause is activated.
      IJogFunctionActive : Bool;   // Jog function is activated.
      IStandbyFunctionDeactivated : Bool;   // Standby function is deactivated.
      WStanbyIsActive : Bool;   // Standby is active and the machine can start by it self.
      WWarningFromHSM_Side : Bool;   // Warning from Side HSM.
      WWarningFromHSM_Zon1 : Bool;   // Warning from Zone 1 HSM.
      WWarningFromHSM_Zon2 : Bool;   // Warning from Zone 2 HSM.
      ATop_Side_HSM_Move_Error : Bool;   // Fault Zone 1 Label adjust motor.
      IEmptyMachineRunning : Bool;   // Machine will run until there's no more products and stop.
      ALowAirPressure : Bool;   // Low air pressure check air and air pressure.
      ICam1Deactivated : Bool;   // Camera 1 deactivated.
      ICam2Deactivated : Bool;   // Camera 2 deactivated.
      ICam3Deactivated : Bool;   // Camera 3 deactivated.
      ICam4Deactivated : Bool;   // Camera 4 deactivated.
      IHSMSideDeactivated : Bool;   // HSM Side deactivated.
      IHSMZone1Deactivated : Bool;   // HSM Zone 1 deactivated.
      IHSMZone2Deactivated : Bool;   // HSM Zone 2 deactivated.
      WSideRejectFull : Bool;   // Reject låda till banderoll full
      ACam1_Max_Rejects_Reached : Bool;   // Camera 1 max rejects reached. Check Camera HMI.
      ISpeed_1 : Bool;   // Speed 1 selected.
      ISpeed_2 : Bool;   // Speed 2 Selected.
      ISpeed_3 : Bool;   // Speed 3 Selected.
      ISpeed_4 : Bool;   // Speed 4 Selected.
      ISpeed_5 : Bool;   // Speed 5 Selected.
      ABufferConveyorFault : Bool;   // Engine protection tripped on buffer conveyor.
      AAC_NotReady : Bool;   // 4050AC is not ready.
      WAC_Warning : Bool;   // Warning from 4050AC.
      IIndexWheelHoming : Bool;   // Index Wheel homing or waiting for products to start homing.
      APrinterNotReady : Bool;   // Printer is not ready
      IPrinterDeactivated : Bool;   // Printer deactivated
      MachineSpeed : Real := 50.0;
   END_VAR
BEGIN
END_DATA_BLOCK

DATA_BLOCK "DB - From_PC"   // DB22
{ S7_Optimized_Access := 'FALSE' }
VERSION : 0.1
// stored: AutoNumber true, DBAccessibleFromOPCUA true, DBAccessibleFromWebserver true, IsOnlyStoredInLoadMemory false, IsWriteProtectedInAS false
   VAR
      WatchDog : Bool;
      Start : Bool;
      Reset : Bool;
      OpenDoor : Bool;
      SnabbStop : Bool;
      ActiveUnwinder : Bool;
      LabelSeamed : Bool;
      Labeler_On : Bool;
      PrinterReady : Bool;
      ShowHMI : Bool;
      LoggedInLevel1 : Bool;
      LoggedInLevel2 : Bool;
      LoggedInLevel3 : Bool;
      BufferConveyor : Bool;
      Stopp : Bool;
   END_VAR
BEGIN
END_DATA_BLOCK

DATA_BLOCK "DB - Motion_Settings"   // DB45
{ S7_Optimized_Access := 'FALSE' }
VERSION : 0.1
// stored: AutoNumber true, DBAccessibleFromOPCUA true, DBAccessibleFromWebserver true, IsOnlyStoredInLoadMemory false, IsWriteProtectedInAS false
   VAR RETAIN
      SideMotionSettings : Struct
         FeedLabelDistance : LReal := -700.0;
         FeedLabelVelocity : LReal := 2000.0;
         FeedLabelAcceleration : LReal := 30000.0;
         FeedLabelDeceleration : LReal := 30000.0;
         FeedLabelJerk : LReal := 1000000.0;
         DispenseLabelDistance : LReal := -675.0;
         DispenseLabelVelocity : LReal := 3000.0;
         DispenseLabelAcceleration : LReal := 500000.0;
         DispenseLabelDeceleration : LReal := 500000.0;
         DispenseLabelJerk : LReal := 5000000.0;
         DispenseLabelJerk_Stop : LReal := 5000000.0;
         DispenseLabelSensorCalibrationDistance : LReal := -84.0;
         RotateProductDistance : LReal := 900.0;
         RotateProductVelocity : LReal := -3000.0;
         RotateProductAcceleration : LReal := 50000.0;
         RotateProductDeceleration : LReal := 35000.0;
         RotateProductJerk : LReal := 2500000.0;
         IndexWheelDistance : LReal := -900.0;
         IndexWheelVelocity : LReal := 18000.0;
         IndexWheelAcceleration : LReal := 50000.0;
         IndexWheelDeceleration : LReal := 50000.0;
         IndexWheelJerk : LReal := 5000000.0;
         RewinderAcceleration : LReal := 20000.0;
         RewinderDeceleration : LReal := 30000.0;
         RewinderJerk : LReal := 2000000.0;
         RewinderPIDSetPoint : Real := 20.0;
         RewinderPIDGain : Real := 1.5;
         RewinderPIDIntegrationTime : Time := T#20s;
         RewinderPIDDeadZone : Real := 1.0;
         RewinderPIDOutputFactor : Real := 30.0;
      END_STRUCT;
      Zon1MotionSettings : Struct
         ConveyorVelocity : LReal := -1395.0;
         QueueVelocity : LReal := 140.0;
         SideHSMVelocity : LReal := 210.0;
         RotationRightRunningVelocity : LReal := 1500.0;
         RotationLeftRunningVelocity : LReal := -1500.0;
      END_STRUCT;
      Zon2MotionSettings : Struct
         ConveyorVelocity : LReal := -1395.0;
         QueueVelocity : LReal := -140.0;
         SideHSMVelocity : LReal := -210.0;
      END_STRUCT;
   END_VAR
BEGIN
END_DATA_BLOCK

DATA_BLOCK "DB - Settings_From_PC"   // DB63
{ S7_Optimized_Access := 'FALSE' }
VERSION : 0.1
// stored: AutoNumber true, DBAccessibleFromOPCUA true, DBAccessibleFromWebserver true, IsOnlyStoredInLoadMemory false, IsWriteProtectedInAS false
   VAR RETAIN
      DispenseLabelSensorCalibration : LReal := 200.0;   // Avstånd från Gap givare till tunga
      SpeedDifferenceDispenser : LReal := -5.0;   // Hastighetsskillnad Dispensering
      DispenseLabelDistance : LReal := -610.0;   // Etikettlängd
      IndexWheel_HomingDistance : LReal := -510.0;   // Indexhjul homing avstånd
      SpeedDifferenceDispeningSplice : LReal := 0.0;   // Hastighetsskillnad Dispensering Start
      PercentageToChangeLabelPosition : LReal := 1.0;   // Procent att ändra etikettposition
      NumberOfRejectsToIgnore : LReal := 20.0;   // Antal underkända dosor att ignorera
      NumberOfProductsBeforeAdjustStart : LReal := 4.0;   // Antal dosor innan justering vid start
      NumberOfProductsBeforeAdjustStop : LReal := 5.0;   // Antal dosor innan justering
      RotateProductMPerMinToDegreesPerSecondCalibrationValue : LReal := 48.0;   // Rotera product motor kalibreringsvärde
      SideRejectDelay : LReal := 0.0;   // Banderoll reject fördröjning
      OrientationValue : LReal := 0.0;   // Orienteringsmotorer kalibrerings värde
      OrientaionCorrectionValue : LReal := 0.0;   // Orintering korrigeringsvärde
      SideSyncLength : LReal;
   END_VAR
BEGIN
END_DATA_BLOCK

DATA_BLOCK "DB - Speed_1"   // DB88
{ S7_Optimized_Access := 'FALSE' }
VERSION : 0.1
// stored: AutoNumber true, DBAccessibleFromOPCUA true, DBAccessibleFromWebserver true, IsOnlyStoredInLoadMemory false, IsWriteProtectedInAS false
   VAR RETAIN
      SpeedSettings : "Speed_Change_Parameters";
   END_VAR
BEGIN
   SpeedSettings.LabelSpeed := 20;
   SpeedSettings.IndexWheelVelocity := 2000.0;
   SpeedSettings.IndexWheelAcceleration := 10000.0;
   SpeedSettings.IndexWheelDeceleration := 10000.0;
   SpeedSettings.IndexWheelJerk := 500000.0;
END_DATA_BLOCK

DATA_BLOCK "DB - Speed_2"   // DB89
{ S7_Optimized_Access := 'FALSE' }
VERSION : 0.1
// stored: AutoNumber true, DBAccessibleFromOPCUA true, DBAccessibleFromWebserver true, IsOnlyStoredInLoadMemory false, IsWriteProtectedInAS false
   VAR RETAIN
      SpeedSettings : "Speed_Change_Parameters";
   END_VAR
BEGIN
   SpeedSettings.LabelSpeed := 25;
   SpeedSettings.IndexWheelVelocity := 3000.0;
   SpeedSettings.IndexWheelAcceleration := 50000.0;
   SpeedSettings.IndexWheelDeceleration := 50000.0;
   SpeedSettings.IndexWheelJerk := 500000.0;
END_DATA_BLOCK

DATA_BLOCK "DB - Speed_3"   // DB90
{ S7_Optimized_Access := 'FALSE' }
VERSION : 0.1
// stored: AutoNumber true, DBAccessibleFromOPCUA true, DBAccessibleFromWebserver true, IsOnlyStoredInLoadMemory false, IsWriteProtectedInAS false
   VAR RETAIN
      SpeedSettings : "Speed_Change_Parameters";
   END_VAR
BEGIN
   SpeedSettings.LabelSpeed := 30;
   SpeedSettings.IndexWheelVelocity := 5000.0;
   SpeedSettings.IndexWheelAcceleration := 100000.0;
   SpeedSettings.IndexWheelDeceleration := 100000.0;
   SpeedSettings.IndexWheelJerk := 1000000.0;
END_DATA_BLOCK

DATA_BLOCK "DB - Speed_4"   // DB101
{ S7_Optimized_Access := 'FALSE' }
VERSION : 0.1
// stored: AutoNumber true, DBAccessibleFromOPCUA true, DBAccessibleFromWebserver true, IsOnlyStoredInLoadMemory false, IsWriteProtectedInAS false
   VAR RETAIN
      SpeedSettings : "Speed_Change_Parameters";
   END_VAR
BEGIN
   SpeedSettings.LabelSpeed := 45;
   SpeedSettings.IndexWheelVelocity := 5000.0;
   SpeedSettings.IndexWheelAcceleration := 100000.0;
   SpeedSettings.IndexWheelDeceleration := 100000.0;
   SpeedSettings.IndexWheelJerk := 1500000.0;
END_DATA_BLOCK

DATA_BLOCK "DB - Speed_5"   // DB102
{ S7_Optimized_Access := 'FALSE' }
VERSION : 0.1
// stored: AutoNumber true, DBAccessibleFromOPCUA true, DBAccessibleFromWebserver true, IsOnlyStoredInLoadMemory false, IsWriteProtectedInAS false
   VAR RETAIN
      SpeedSettings : "Speed_Change_Parameters";
   END_VAR
BEGIN
   SpeedSettings.LabelSpeed := 60;
   SpeedSettings.IndexWheelVelocity := 10000.0;
   SpeedSettings.IndexWheelAcceleration := 150000.0;
   SpeedSettings.IndexWheelDeceleration := 150000.0;
   SpeedSettings.IndexWheelJerk := 3000000.0;
END_DATA_BLOCK

DATA_BLOCK "DB - To_PC"   // DB23
{ S7_Optimized_Access := 'FALSE' }
VERSION : 0.1
// stored: AutoNumber true, DBAccessibleFromOPCUA true, DBAccessibleFromWebserver true, IsOnlyStoredInLoadMemory false, IsWriteProtectedInAS false
   VAR
      WatchDog : Bool;
      Start : Bool;
      Reset : Bool;
      Door : Bool;
      SnabbStopp : Bool;
      NeedReset : Bool;
      StopToPC : Bool;
      LabelSeamed : Bool;
      Starting : Bool;
      Stopping : Bool;
      Labeler_On : Bool;
      ShowHMI : Bool;
      BufferConveyor : Bool;
   END_VAR
BEGIN
END_DATA_BLOCK

DATA_BLOCK "DB_Statistics_Com"   // DB1
{ S7_Optimized_Access := 'FALSE' }
VERSION : 0.1
// stored: AutoNumber true, DBAccessibleFromOPCUA true, DBAccessibleFromWebserver true, IsOnlyStoredInLoadMemory false, IsWriteProtectedInAS false
   VAR
      Stat : "UDT_Subsystem_Utility";
   END_VAR
BEGIN
END_DATA_BLOCK

DATA_BLOCK "DB - 05_Alarms_From_HSM"   // DB550
{ S7_Optimized_Access := 'FALSE' }
VERSION : 0.1
// stored: AutoNumber false, DBAccessibleFromOPCUA true, DBAccessibleFromWebserver true, IsOnlyStoredInLoadMemory false, IsWriteProtectedInAS false
   VAR
      HSM1 : "HSM_AlarmWarning";
      HSM2 : "HSM_AlarmWarning";
      HSM3 : "HSM_AlarmWarning";
      iWarning00_From_HSM_X : Int;
      iWarning01_From_HSM_X : Int;
      iWarning02_From_HSM_X : Int;
      iWarning03_From_HSM_X : Int;
      iWarning04_From_HSM_X : Int;
      iWarning05_From_HSM_X : Int;
      iWarning06_From_HSM_X : Int;
      iWarning07_From_HSM_X : Int;
      iWarning08_From_HSM_X : Int;
      iWarning09_From_HSM_X : Int;
      iWarning10_From_HSM_X : Int;
      iWarning11_From_HSM_X : Int;
      iWarning12_From_HSM_X : Int;
      iWarning13_From_HSM_X : Int;
      iWarning14_From_HSM_X : Int;
      iWarning15_From_HSM_X : Int;
      iError00_From_HSM_X : Int;
      iError01_From_HSM_X : Int;
      iError02_From_HSM_X : Int;
      iError03_From_HSM_X : Int;
      iError04_From_HSM_X : Int;
      iError05_From_HSM_X : Int;
      iError06_From_HSM_X : Int;
      iError07_From_HSM_X : Int;
      iError08_From_HSM_X : Int;
      iError09_From_HSM_X : Int;
      iError10_From_HSM_X : Int;
      iError11_From_HSM_X : Int;
      iError12_From_HSM_X : Int;
      iError13_From_HSM_X : Int;
      iError14_From_HSM_X : Int;
      iError15_From_HSM_X : Int;
   END_VAR
BEGIN
END_DATA_BLOCK

DATA_BLOCK "DB - 06_Errors_And_Warnings_HSM"   // DB98
{ S7_Optimized_Access := 'TRUE' }
VERSION : 0.1
// stored: AutoNumber false, DBAccessibleFromOPCUA true, DBAccessibleFromWebserver true, IsOnlyStoredInLoadMemory false, IsRetainMemResEnabled false, IsWriteProtectedInAS false, MemoryReserve 0
   VAR
      Alarm_1_HSM_NotReady_1 : Bool;
      Alarm_2_HSM_PLC_Conn_Faulty_1 : Bool;
      Alarm_3_HSM_NotReady_2 : Bool;
      Alarm_4_HSM_PLC_Conn_Faulty_2 : Bool;
      Alarm_5_HSM_NotReady_3 : Bool;
      Alarm_6_HSM_PLC_Conn_Faulty_3 : Bool;
      Alarm_7_Motor_Start_Error : Bool;
      Alarm_8_Motor_Position_Error : Bool;
      Alarm_9_Motor_Position_Control_Error : Bool;
      Alarm_10_Motor_Current_Target_Not_Reached : Bool;
      Alarm_11_Label_Gap_Not_Found : Bool;
      Alarm_12_Unwinder_Web_Break : Bool;
      Alarm_13_Web_End : Bool;
      Alarm_14_Motor_Overcurrent : Bool;
      Alarm_15_Dancer_Arm_Stop_Reached : Bool;
      Alarm_16 : Bool;
      Alarm_17_Rewinder_Web_Break : Bool;
      Alarm_18 : Bool;
      Alarm_19 : Bool;
      Alarm_20 : Bool;
      Warning_01_Find_Rotor_Position : Bool;
      Warning_02 : Bool;
      Warning_03_Number_Of_Labels_Reached : Bool;
      Warning_04_Low_Label_Reached : Bool;
      Warning_05_ZeroDownTime_Lan_Link_timeout : Bool;
      Warning_06_ZeroDownTime_Parameter_error : Bool;
      Warning_07 : Bool;
      Warning_08 : Bool;
      Warning_09_Roll_End_1 : Bool;
      Warning_10_Roll_End_2 : Bool;
      Warning_11_Roll_End_3 : Bool;
      Warning_10_HSM_1_PLC_DataTransmission_Error : Bool;
      Warning_13_HSM_2_PLC_DataTransmission_Error : Bool;
      Warning_14_HSM_3_PLC_DataTransmission_Error : Bool;
   END_VAR
BEGIN
END_DATA_BLOCK

DATA_BLOCK "DB - HSM"   // DB18
{ S7_Optimized_Access := 'FALSE' }
VERSION : 0.1
// stored: AutoNumber true, DBAccessibleFromOPCUA true, DBAccessibleFromWebserver true, IsOnlyStoredInLoadMemory false, IsWriteProtectedInAS false
   VAR RETAIN
      HSM_Side : "typeFromHMI";
      HSM_Zon1 : "typeFromHMI";
      HSM_Zon2_SideTaxStamp : "typeFromHMI";
      xDisable_Parameter_Update_HSM_Side : Bool;   // Disable update parameter changes
      xDisable_Parameter_Update_HSM_Zon1 : Bool;   // Disable update parameter changes
      xDisable_Parameter_Update_HSM_Zon2 : Bool;   // Disable update parameter changes
   END_VAR
BEGIN
   HSM_Side.rLabel_Speed := 28.0;
   HSM_Side.xBtn_Save_Par := false;
   HSM_Side.xHSM_Active := TRUE;
   HSM_Side.xGet_Parameters := false;
   HSM_Side.iLabels_Per_Trigger := 1;
   HSM_Side.iTrigger_Supression := 0;
   HSM_Side.iProduct_Sensor_Polarity := 3;
   HSM_Side.iDouble_Label := 0;
   HSM_Side.iSpeed_Int_Ext := 1;
   HSM_Side.iLabel_Length := 0;
   HSM_Side.rLabel_Position := 1.0;
   HSM_Side.rTrig_Delay := 0.0;
   HSM_Side.rSpeed_Offset := 0.0;
   HSM_Side.rGap_Sensor_To_Dispenser_Tongue := 245.0;
   HSM_Side.rLabel_Spacing := 2.0;
   HSM_Side.rPre_Dispensing_Lenght := 0.0;
   HSM_Side.rLabel_Gap := 0.0;
   HSM_Side.ConfigAndMachineParaMask.HSMConfig_1.iDesiredInternalSpeed := true;
   HSM_Side.ConfigAndMachineParaMask.HSMConfig_1.iDispenseDelay := true;
   HSM_Side.ConfigAndMachineParaMask.HSMMachine_2.iSyncOutputDelay := true;
   HSM_Side.ConfigAndMachineParaMask.HSMMachine_2.iSyncOutputLenght := true;
   HSM_Zon1.rLabel_Speed := 28.0;
   HSM_Zon1.xHSM_Active := TRUE;
   HSM_Zon1.iLabels_Per_Trigger := 1;
   HSM_Zon1.iTrigger_Supression := 0;
   HSM_Zon1.iProduct_Sensor_Polarity := 2;
   HSM_Zon1.iDouble_Label := 0;
   HSM_Zon1.iSpeed_Int_Ext := 1;
   HSM_Zon1.iLabel_Length := 0;
   HSM_Zon1.rLabel_Position := 1.0;
   HSM_Zon1.rTrig_Delay := 0.0;
   HSM_Zon1.rSpeed_Offset := 0.0;
   HSM_Zon1.rGap_Sensor_To_Dispenser_Tongue := 125.0;
   HSM_Zon1.rLabel_Spacing := 2.0;
   HSM_Zon1.rPre_Dispensing_Lenght := 0.0;
   HSM_Zon1.rLabel_Gap := 0.0;
   HSM_Zon1.ConfigAndMachineParaMask.HSMConfig_1.iDesiredInternalSpeed := true;
   HSM_Zon1.ConfigAndMachineParaMask.HSMConfig_1.iDispenseDelay := true;
   HSM_Zon1.ConfigAndMachineParaMask.HSMConfig_1.iLabelPosition := true;
   HSM_Zon2_SideTaxStamp.rLabel_Speed := 28.0;
   HSM_Zon2_SideTaxStamp.xBtn_Save_Par := false;
   HSM_Zon2_SideTaxStamp.xHSM_Active := TRUE;
   HSM_Zon2_SideTaxStamp.xGet_Parameters := false;
   HSM_Zon2_SideTaxStamp.iLabels_Per_Trigger := 1;
   HSM_Zon2_SideTaxStamp.iTrigger_Supression := 0;
   HSM_Zon2_SideTaxStamp.iProduct_Sensor_Polarity := 3;
   HSM_Zon2_SideTaxStamp.iDouble_Label := 0;
   HSM_Zon2_SideTaxStamp.iSpeed_Int_Ext := 1;
   HSM_Zon2_SideTaxStamp.iLabel_Length := 0;
   HSM_Zon2_SideTaxStamp.rLabel_Position := 1.0;
   HSM_Zon2_SideTaxStamp.rTrig_Delay := 0.0;
   HSM_Zon2_SideTaxStamp.rSpeed_Offset := 0.0;
   HSM_Zon2_SideTaxStamp.rGap_Sensor_To_Dispenser_Tongue := 125.0;
   HSM_Zon2_SideTaxStamp.rLabel_Spacing := 2.0;
   HSM_Zon2_SideTaxStamp.rPre_Dispensing_Lenght := 0.0;
   HSM_Zon2_SideTaxStamp.rLabel_Gap := 0.0;
   HSM_Zon2_SideTaxStamp.ConfigAndMachineParaMask.HSMConfig_1.iDesiredInternalSpeed := true;
   HSM_Zon2_SideTaxStamp.ConfigAndMachineParaMask.HSMConfig_1.iDispenseDelay := true;
   HSM_Zon2_SideTaxStamp.ConfigAndMachineParaMask.HSMConfig_1.iLabelPosition := true;
   HSM_Zon2_SideTaxStamp.ConfigAndMachineParaMask.HSMMachine_1.iDistanceToDispensingEdgeToGapSensor := true;
END_DATA_BLOCK

DATA_BLOCK "DB - HSM_Side_From"   // DB55
{ S7_Optimized_Access := 'FALSE' }
VERSION : 0.1
// stored: AutoNumber false, DBAccessibleFromOPCUA true, DBAccessibleFromWebserver true, IsOnlyStoredInLoadMemory false, IsWriteProtectedInAS false
   VAR
      DataFromHSM : "DataFromHSM";
   END_VAR
BEGIN
   // DataFromHSM.Sts : Status From HSM
   // DataFromHSM.Cfg : Configuration Parameters Receive
   // DataFromHSM.M_Par : Machine Parameters Receive
END_DATA_BLOCK

DATA_BLOCK "DB - HSM_Side_To"   // DB53
{ S7_Optimized_Access := 'FALSE' }
VERSION : 0.1
// stored: AutoNumber false, DBAccessibleFromOPCUA true, DBAccessibleFromWebserver true, IsOnlyStoredInLoadMemory false, IsWriteProtectedInAS false
   VAR
      DataToHSM : "DataToHSM";
   END_VAR
BEGIN
END_DATA_BLOCK

DATA_BLOCK "DB - HSM_Zon1_From"   // DB64
{ S7_Optimized_Access := 'FALSE' }
VERSION : 0.1
// stored: AutoNumber false, DBAccessibleFromOPCUA true, DBAccessibleFromWebserver true, IsOnlyStoredInLoadMemory false, IsWriteProtectedInAS false
   VAR
      DataFromHSM : "DataFromHSM";
   END_VAR
BEGIN
   // DataFromHSM.Sts : Status From HSM
   // DataFromHSM.Cfg : Configuration Parameters Receive
   // DataFromHSM.M_Par : Machine Parameters Receive
END_DATA_BLOCK

DATA_BLOCK "DB - HSM_Zon1_To"   // DB59
{ S7_Optimized_Access := 'FALSE' }
VERSION : 0.1
// stored: AutoNumber false, DBAccessibleFromOPCUA true, DBAccessibleFromWebserver true, IsOnlyStoredInLoadMemory false, IsWriteProtectedInAS false
   VAR
      DataToHSM : "DataToHSM";
   END_VAR
BEGIN
END_DATA_BLOCK

DATA_BLOCK "DB - HSM_Zon2_From"   // DB68
{ S7_Optimized_Access := 'FALSE' }
VERSION : 0.1
// stored: AutoNumber false, DBAccessibleFromOPCUA true, DBAccessibleFromWebserver true, IsOnlyStoredInLoadMemory false, IsWriteProtectedInAS false
   VAR
      DataFromHSM : "DataFromHSM";
   END_VAR
BEGIN
   // DataFromHSM.Sts : Status From HSM
   // DataFromHSM.Cfg : Configuration Parameters Receive
   // DataFromHSM.M_Par : Machine Parameters Receive
END_DATA_BLOCK

DATA_BLOCK "DB - HSM_Zon2_To"   // DB69
{ S7_Optimized_Access := 'FALSE' }
VERSION : 0.1
// stored: AutoNumber false, DBAccessibleFromOPCUA true, DBAccessibleFromWebserver true, IsOnlyStoredInLoadMemory false, IsWriteProtectedInAS false
   VAR
      DataToHSM : "DataToHSM";
   END_VAR
BEGIN
END_DATA_BLOCK

ORGANIZATION_BLOCK "Main"   // OB1, LAD, ProgramCycle
TITLE = "Main Program Sweep (Cycle)"
{ S7_Optimized_Access := 'TRUE' }
VERSION : 0.1
// stored: AutoNumber true, IsIECCheckEnabled false, SetENOAutomatically false
   VAR_INPUT
      Initial_Call : Bool;   // Initial call of this OB
      Remanence : Bool;   // =True, if remanent data are available
   END_VAR
BEGIN

REGION Network 1
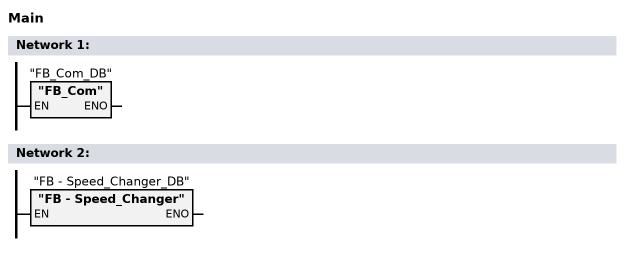
   RUNG wire#powerrail
      "FB_Com_DB"()
   END_RUNG
   // the same network as SCL:
   "FB_Com_DB"();   // "FB_Com"
END_REGION

REGION Network 2
   RUNG wire#powerrail
      "FB - Speed_Changer_DB"()
   END_RUNG
   // the same network as SCL:
   "FB - Speed_Changer_DB"();   // "FB - Speed_Changer"
END_REGION
END_ORGANIZATION_BLOCK

FUNCTION_BLOCK "FB_Com"   // FB1, LAD
{ S7_Optimized_Access := 'TRUE' }
VERSION : 0.1
// stored: AutoNumber true, IsIECCheckEnabled false, IsRetainMemResEnabled false, MemoryReserve 100, SetENOAutomatically false, UDAEnableTagReadback false
   VAR
      TRCV_C_Instance { S7_SetPoint := 'True'} : TRCV_C;
      GET_Instance { S7_SetPoint := 'True'} : GET;
      TRCV_C_Instance_1 { S7_SetPoint := 'True'} : TRCV_C;
      Diff : LInt;
   END_VAR
BEGIN

REGION Network 1
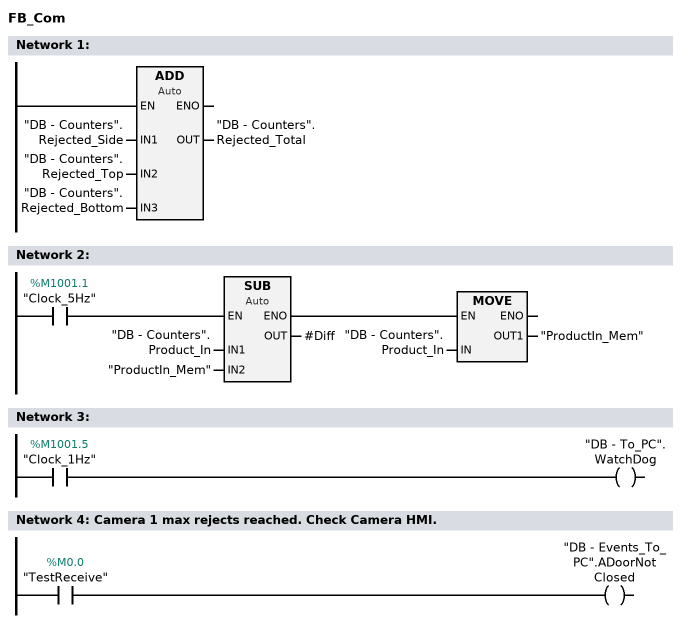
   RUNG wire#powerrail
      Add(in1 := "DB - Counters".Rejected_Side, in2 := "DB - Counters".Rejected_Top, in3 := "DB - Counters".Rejected_Bottom, out => "DB - Counters".Rejected_Total)
   END_RUNG
   // the same network as SCL:
   "DB - Counters".Rejected_Total := "DB - Counters".Rejected_Side + "DB - Counters".Rejected_Top + "DB - Counters".Rejected_Bottom;
END_REGION

REGION Network 2
   RUNG wire#powerrail
      Contact( "Clock_5Hz" )
      Sub(in1 := "DB - Counters".Product_In, in2 := "ProductIn_Mem", out => #Diff)
      Move(in := "DB - Counters".Product_In, out1 => "ProductIn_Mem")
   END_RUNG
   // the same network as SCL:
   IF "Clock_5Hz" THEN
       #Diff := "DB - Counters".Product_In - "ProductIn_Mem";
       "ProductIn_Mem" := "DB - Counters".Product_In;
   END_IF;
END_REGION

REGION Network 3
   RUNG wire#powerrail
      Contact( "Clock_1Hz" )
      Coil( "DB - To_PC".WatchDog )
   END_RUNG
   // the same network as SCL:
   "DB - To_PC".WatchDog := "Clock_1Hz";
END_REGION

REGION Network 4: Camera 1 max rejects reached. Check Camera HMI.
   RUNG wire#powerrail
      Contact( "TestReceive" )
      Coil( "DB - Events_To_PC".ADoorNotClosed )
   END_RUNG
   // the same network as SCL:
   "DB - Events_To_PC".ADoorNotClosed := "TestReceive";
END_REGION
END_FUNCTION_BLOCK

FUNCTION_BLOCK "FB - Speed_Changer"   // FB37, LAD
{ S7_Optimized_Access := 'TRUE' }
VERSION : 0.1
// stored: AutoNumber true, IsIECCheckEnabled false, IsRetainMemResEnabled false, MemoryReserve 100, SetENOAutomatically false, UDAEnableTagReadback false
   VAR
      Speed_1_Pos : Bool;
      Speed_2_Pos : Bool;
      Speed_3_Pos : Bool;
      Speed_4_Pos : Bool;
      IEC_Timer_0_Instance { S7_SetPoint := 'True'} : TON_TIME;
      ResetSpeedEvents : Bool;
      Speed_5_Pos : Bool;
   END_VAR
   VAR_TEMP   // added for the SCL form of the ladder/FBD networks
      _w1 : Bool;
   END_VAR
BEGIN

REGION Network 1: Reset Speed Tags
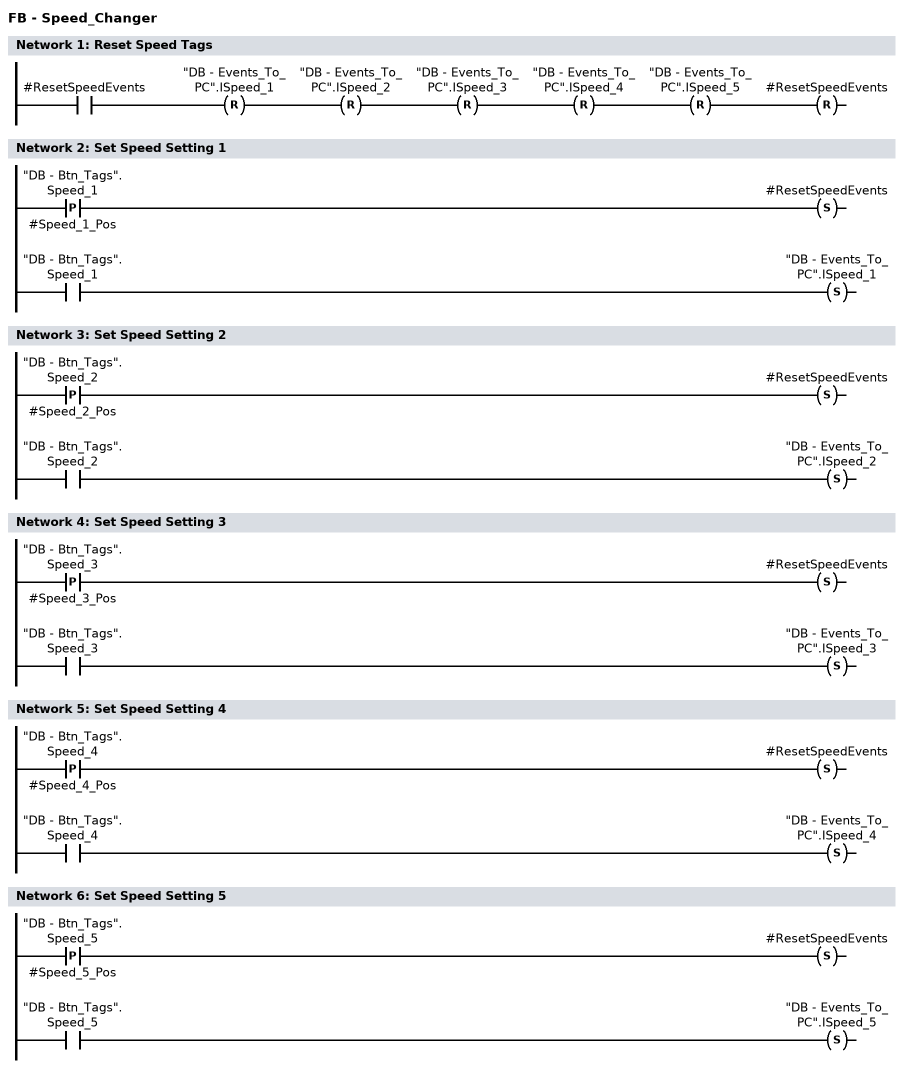
   RUNG wire#powerrail
      Contact( #ResetSpeedEvents )
      R_Coil( "DB - Events_To_PC".ISpeed_1 )
      R_Coil( "DB - Events_To_PC".ISpeed_2 )
      R_Coil( "DB - Events_To_PC".ISpeed_3 )
      R_Coil( "DB - Events_To_PC".ISpeed_4 )
      R_Coil( "DB - Events_To_PC".ISpeed_5 )
      R_Coil( #ResetSpeedEvents )
   END_RUNG
   // the same network as SCL:
   IF #ResetSpeedEvents THEN
       "DB - Events_To_PC".ISpeed_1 := FALSE;
       "DB - Events_To_PC".ISpeed_2 := FALSE;
       "DB - Events_To_PC".ISpeed_3 := FALSE;
       "DB - Events_To_PC".ISpeed_4 := FALSE;
       "DB - Events_To_PC".ISpeed_5 := FALSE;
       #ResetSpeedEvents := FALSE;
   END_IF;
END_REGION

REGION Network 2: Set Speed Setting 1
   RUNG wire#powerrail
      P_Contact(operand := "DB - Btn_Tags".Speed_1, bit := #Speed_1_Pos)
      S_Coil( #ResetSpeedEvents )
   END_RUNG
   RUNG wire#powerrail
      Contact( "DB - Btn_Tags".Speed_1 )
      S_Coil( "DB - Events_To_PC".ISpeed_1 )
   END_RUNG
   // the same network as SCL:
   #_w1 := "DB - Btn_Tags".Speed_1 AND NOT #Speed_1_Pos;   // rising edge of "DB - Btn_Tags".Speed_1
   #Speed_1_Pos := "DB - Btn_Tags".Speed_1;
   IF #_w1 THEN #ResetSpeedEvents := TRUE; END_IF;
   IF "DB - Btn_Tags".Speed_1 THEN "DB - Events_To_PC".ISpeed_1 := TRUE; END_IF;
END_REGION

REGION Network 3: Set Speed Setting 2
   RUNG wire#powerrail
      P_Contact(operand := "DB - Btn_Tags".Speed_2, bit := #Speed_2_Pos)
      S_Coil( #ResetSpeedEvents )
   END_RUNG
   RUNG wire#powerrail
      Contact( "DB - Btn_Tags".Speed_2 )
      S_Coil( "DB - Events_To_PC".ISpeed_2 )
   END_RUNG
   // the same network as SCL:
   #_w1 := "DB - Btn_Tags".Speed_2 AND NOT #Speed_2_Pos;   // rising edge of "DB - Btn_Tags".Speed_2
   #Speed_2_Pos := "DB - Btn_Tags".Speed_2;
   IF #_w1 THEN #ResetSpeedEvents := TRUE; END_IF;
   IF "DB - Btn_Tags".Speed_2 THEN "DB - Events_To_PC".ISpeed_2 := TRUE; END_IF;
END_REGION

REGION Network 4: Set Speed Setting 3
   RUNG wire#powerrail
      P_Contact(operand := "DB - Btn_Tags".Speed_3, bit := #Speed_3_Pos)
      S_Coil( #ResetSpeedEvents )
   END_RUNG
   RUNG wire#powerrail
      Contact( "DB - Btn_Tags".Speed_3 )
      S_Coil( "DB - Events_To_PC".ISpeed_3 )
   END_RUNG
   // the same network as SCL:
   #_w1 := "DB - Btn_Tags".Speed_3 AND NOT #Speed_3_Pos;   // rising edge of "DB - Btn_Tags".Speed_3
   #Speed_3_Pos := "DB - Btn_Tags".Speed_3;
   IF #_w1 THEN #ResetSpeedEvents := TRUE; END_IF;
   IF "DB - Btn_Tags".Speed_3 THEN "DB - Events_To_PC".ISpeed_3 := TRUE; END_IF;
END_REGION

REGION Network 5: Set Speed Setting 4
   RUNG wire#powerrail
      P_Contact(operand := "DB - Btn_Tags".Speed_4, bit := #Speed_4_Pos)
      S_Coil( #ResetSpeedEvents )
   END_RUNG
   RUNG wire#powerrail
      Contact( "DB - Btn_Tags".Speed_4 )
      S_Coil( "DB - Events_To_PC".ISpeed_4 )
   END_RUNG
   // the same network as SCL:
   #_w1 := "DB - Btn_Tags".Speed_4 AND NOT #Speed_4_Pos;   // rising edge of "DB - Btn_Tags".Speed_4
   #Speed_4_Pos := "DB - Btn_Tags".Speed_4;
   IF #_w1 THEN #ResetSpeedEvents := TRUE; END_IF;
   IF "DB - Btn_Tags".Speed_4 THEN "DB - Events_To_PC".ISpeed_4 := TRUE; END_IF;
END_REGION

REGION Network 6: Set Speed Setting 5
   RUNG wire#powerrail
      P_Contact(operand := "DB - Btn_Tags".Speed_5, bit := #Speed_5_Pos)
      S_Coil( #ResetSpeedEvents )
   END_RUNG
   RUNG wire#powerrail
      Contact( "DB - Btn_Tags".Speed_5 )
      S_Coil( "DB - Events_To_PC".ISpeed_5 )
   END_RUNG
   // the same network as SCL:
   #_w1 := "DB - Btn_Tags".Speed_5 AND NOT #Speed_5_Pos;   // rising edge of "DB - Btn_Tags".Speed_5
   #Speed_5_Pos := "DB - Btn_Tags".Speed_5;
   IF #_w1 THEN #ResetSpeedEvents := TRUE; END_IF;
   IF "DB - Btn_Tags".Speed_5 THEN "DB - Events_To_PC".ISpeed_5 := TRUE; END_IF;
END_REGION
END_FUNCTION_BLOCK

DATA_BLOCK "FB - Speed_Changer_DB"   // DB4
VERSION : 0.1
// stored: AutoNumber true, DBAccessibleFromOPCUA true, DBAccessibleFromWebserver true, InstanceOfName FB - Speed_Changer, InstanceOfType FB
"FB - Speed_Changer"
BEGIN
END_DATA_BLOCK

DATA_BLOCK "FB_Com_DB"   // DB3
VERSION : 0.1
// stored: AutoNumber true, DBAccessibleFromOPCUA true, DBAccessibleFromWebserver true, InstanceOfName FB_Com, InstanceOfType FB
"FB_Com"
BEGIN
END_DATA_BLOCK
